LIN {X 0,Y 516.034,Z 964.883,A -85,B 0,C 180,E1 13801.811,E2 13801.811} C_VEL
LIN {X 0,Y 525.907,Z 921.872,A -85,B 0,C 180,E1 13804.841,E2 13804.841} C_VEL
LIN {X 0,Y 533.905,Z 879.595,A -85,B 0,C 180,E1 13807.015,E2 13807.015} C_VEL
LIN {X 0,Y 536.579,Z 858.24,A -85,B 0,C 180,E1 13807.941,E2 13807.941} C_VEL
LIN {X 0,Y 518.339,Z 819.478,A -85,B 0,C 180,E1 13812.064,E2 13812.064} C_VEL
LIN {X 0,Y 498.945,Z 786.831,A -85,B 0,C 180,E1 13816.041,E2 13816.041} C_VEL
LIN {X 0,Y 481.398,Z 761.941,A -85,B 0,C 180,E1 13819.773,E2 13819.773} C_VEL
LIN {X 0,Y 477.173,Z 755.892,A -85,B 0,C 180,E1 13820.762,E2 13820.762} C_VEL
LIN {X 0,Y 474.157,Z 751.123,A -85,B 0,C 180,E1 13821.51,E2 13821.51} C_VEL
LIN {X 0,Y 474.006,Z 749.56,A -85,B 0,C 180,E1 13821.607,E2 13821.607} C_VEL
LIN {X 0,Y 473.918,Z 749.56,A -85,B 0,C 180,E1 13827.169,E2 13827.169} C_VEL
LIN {X 0,Y 474.069,Z 749.56,A -85,B 0,C 180,E1 13833.49,E2 13833.49} C_VEL
LIN {X 0,Y 474.276,Z 749.56,A -85,B 0,C 180,E1 13839.477,E2 13839.477} C_VEL
LIN {X 0,Y 474.538,Z 749.56,A -85,B 0,C 180,E1 13845.235,E2 13845.235} C_VEL
LIN {X 0,Y 475.007,Z 749.56,A -85,B 0,C 180,E1 13850.842,E2 13850.842} C_VEL
LIN {X 0,Y 475.371,Z 749.56,A -85,B 0,C 180,E1 13856.35,E2 13856.35} C_VEL
LIN {X 0,Y 475.462,Z 749.56,A -85,B 0,C 180,E1 13861.816,E2 13861.816} C_VEL
LIN {X 0,Y 475.102,Z 749.56,A -85,B 0,C 180,E1 13867.304,E2 13867.304} C_VEL
LIN {X 0,Y 474.846,Z 749.56,A -85,B 0,C 180,E1 13872.867,E2 13872.867} C_VEL
LIN {X 0,Y 474.618,Z 749.56,A -85,B 0,C 180,E1 13878.561,E2 13878.561} C_VEL
LIN {X 0,Y 474.385,Z 750.237,A -85,B 0,C 180,E1 13884.27,E2 13884.27} C_VEL
LIN {X 0,Y 477.004,Z 755.483,A -85,B 0,C 180,E1 13884.954,E2 13884.954} C_VEL
LIN {X 0,Y 479.513,Z 758.583,A -85,B 0,C 180,E1 13885.535,E2 13885.535} C_VEL
LIN {X 0,Y 500.029,Z 787.996,A -85,B 0,C 180,E1 13889.906,E2 13889.906} C_VEL
LIN {X 0,Y 523.015,Z 825.421,A -85,B 0,C 180,E1 13894.162,E2 13894.162} C_VEL
LIN {X 0,Y 542.914,Z 863.835,A -85,B 0,C 180,E1 13897.881,E2 13897.881} C_VEL
LIN {X 0,Y 544.784,Z 869.388,A -85,B 0,C 180,E1 13898.295,E2 13898.295} C_VEL
LIN {X 0,Y 537.645,Z 917.442,A -85,B 0,C 180,E1 13899.901,E2 13899.901} C_VEL
LIN {X 0,Y 529.329,Z 963.938,A -85,B 0,C 180,E1 13902.158,E2 13902.158} C_VEL
LIN {X 0,Y 519.683,Z 1007.812,A -85,B 0,C 180,E1 13905.042,E2 13905.042} C_VEL
LIN {X 0,Y 509.605,Z 1048.714,A -85,B 0,C 180,E1 13908.52,E2 13908.52} C_VEL
LIN {X 0,Y 499.79,Z 1087.044,A -85,B 0,C 180,E1 13912.791,E2 13912.791} C_VEL
LIN {X 0,Y 491.205,Z 1120.824,A -85,B 0,C 180,E1 13917.595,E2 13917.595} C_VEL
LIN {X 0,Y 484.254,Z 1149.865,A -85,B 0,C 180,E1 13922.926,E2 13922.926} C_VEL
LIN {X 0,Y 479.949,Z 1171.932,A -85,B 0,C 180,E1 13928.124,E2 13928.124} C_VEL
LIN {X 0,Y 477.25,Z 1188.833,A -85,B 0,C 180,E1 13933.442,E2 13933.442} C_VEL
LIN {X 0,Y 475.934,Z 1200.642,A -85,B 0,C 180,E1 13939.017,E2 13939.017} C_VEL
LIN {X 0,Y 475.666,Z 1203.715,A -85,B 0,C 180,E1 13941.011,E2 13941.011} C_VEL
LIN {X 0,Y 473.053,Z 1205.774,A -85,B 0,C 180,E1 13942.541,E2 13942.541} C_VEL
LIN {X 0,Y 467.534,Z 1208.179,A -85,B 0,C 180,E1 13945.048,E2 13945.048} C_VEL
LIN {X 0,Y 467.525,Z 1208.086,A -85,B 0,C 180,E1 13945.115,E2 13945.115} C_VEL
LIN {X 0,Y 467.648,Z 1210,A -85,B 0,C 180,E1 13949.999,E2 13949.999} C_VEL
LIN {X 0,Y 467.584,Z 1207.633,A -85,B 0,C 180,E1 13955.563,E2 13955.563} C_VEL
LIN {X 0,Y 468.047,Z 1200.643,A -85,B 0,C 180,E1 13961.169,E2 13961.169} C_VEL
LIN {X 0,Y 469.297,Z 1189.506,A -85,B 0,C 180,E1 13966.364,E2 13966.364} C_VEL
LIN {X 0,Y 471.984,Z 1172.687,A -85,B 0,C 180,E1 13971.811,E2 13971.811} C_VEL
LIN {X 0,Y 476.377,Z 1150.561,A -85,B 0,C 180,E1 13977.183,E2 13977.183} C_VEL
LIN {X 0,Y 483.69,Z 1120.879,A -85,B 0,C 180,E1 13982.724,E2 13982.724} C_VEL
LIN {X 0,Y 492.65,Z 1086.82,A -85,B 0,C 180,E1 13987.664,E2 13987.664} C_VEL
LIN {X 0,Y 503.17,Z 1048.376,A -85,B 0,C 180,E1 13992.052,E2 13992.052} C_VEL
LIN {X 0,Y 514.127,Z 1007.233,A -85,B 0,C 180,E1 13995.657,E2 13995.657} C_VEL
LIN {X 0,Y 524.703,Z 963.33,A -85,B 0,C 180,E1 13998.628,E2 13998.628} C_VEL
LIN {X 0,Y 534.281,Z 915.858,A -85,B 0,C 180,E1 14000.977,E2 14000.977} C_VEL
LIN {X 0,Y 541.086,Z 870.88,A -85,B 0,C 180,E1 14002.601,E2 14002.601} C_VEL
LIN {X 0,Y 528.086,Z 840.131,A -85,B 0,C 180,E1 14005.85,E2 14005.85} C_VEL
LIN {X 0,Y 513.151,Z 814.352,A -85,B 0,C 180,E1 14009.429,E2 14009.429} C_VEL
LIN {X 0,Y 497.416,Z 791.232,A -85,B 0,C 180,E1 14013.626,E2 14013.626} C_VEL
LIN {X 0,Y 486.968,Z 777.414,A -85,B 0,C 180,E1 14016.94,E2 14016.94} C_VEL
LIN {X 0,Y 482.346,Z 771.07,A -85,B 0,C 180,E1 14018.647,E2 14018.647} C_VEL
LIN {X 0,Y 478.295,Z 764.996,A -85,B 0,C 180,E1 14020.33,E2 14020.33} C_VEL
LIN {X 0,Y 473.236,Z 759.393,A -85,B 0,C 180,E1 14022.628,E2 14022.628} C_VEL
LIN {X 0,Y 472.102,Z 757.06,A -85,B 0,C 180,E1 14023.262,E2 14023.262} C_VEL
LIN {X 0,Y 467.454,Z 752.711,A -85,B 0,C 180,E1 14025.88,E2 14025.88} C_VEL
LIN {X 0,Y 466.84,Z 749.56,A -85,B 0,C 180,E1 14026.622,E2 14026.622} C_VEL
LIN {X 0,Y 467.194,Z 749.56,A -85,B 0,C 180,E1 14032.571,E2 14032.571} C_VEL
LIN {X 0,Y 467.541,Z 749.56,A -85,B 0,C 180,E1 14038.153,E2 14038.153} C_VEL
LIN {X 0,Y 467.467,Z 749.56,A -85,B 0,C 180,E1 14043.712,E2 14043.712} C_VEL
LIN {X 0,Y 467.127,Z 750.157,A -85,B 0,C 180,E1 14049.255,E2 14049.255} C_VEL
LIN {X 0,Y 469.125,Z 754.964,A -85,B 0,C 180,E1 14050.679,E2 14050.679} C_VEL
LIN {X 0,Y 472.981,Z 758.131,A -85,B 0,C 180,E1 14052.694,E2 14052.694} C_VEL
LIN {X 0,Y 476.564,Z 763.704,A -85,B 0,C 180,E1 14054.466,E2 14054.466} C_VEL
LIN {X 0,Y 478.873,Z 766.162,A -85,B 0,C 180,E1 14055.447,E2 14055.447} C_VEL
LIN {X 0,Y 483.501,Z 771.831,A -85,B 0,C 180,E1 14057.278,E2 14057.278} C_VEL
LIN {X 0,Y 495.775,Z 789.143,A -85,B 0,C 180,E1 14061.46,E2 14061.46} C_VEL
LIN {X 0,Y 509.693,Z 809.728,A -85,B 0,C 180,E1 14065.505,E2 14065.505} C_VEL
LIN {X 0,Y 524.946,Z 837.122,A -85,B 0,C 180,E1 14069.707,E2 14069.707} C_VEL
LIN {X 0,Y 536.072,Z 863.906,A -85,B 0,C 180,E1 14073.041,E2 14073.041} C_VEL
LIN {X 0,Y 527.801,Z 907.851,A -85,B 0,C 180,E1 14075.105,E2 14075.105} C_VEL
LIN {X 0,Y 517.224,Z 951.582,A -85,B 0,C 180,E1 14077.925,E2 14077.925} C_VEL
LIN {X 0,Y 506.236,Z 989.958,A -85,B 0,C 180,E1 14081.275,E2 14081.275} C_VEL
LIN {X 0,Y 495.534,Z 1024.827,A -85,B 0,C 180,E1 14085.28,E2 14085.28} C_VEL
LIN {X 0,Y 485.435,Z 1057.02,A -85,B 0,C 180,E1 14090.171,E2 14090.171} C_VEL
LIN {X 0,Y 477.545,Z 1083.26,A -85,B 0,C 180,E1 14095.49,E2 14095.49} C_VEL
LIN {X 0,Y 472.449,Z 1103.182,A -85,B 0,C 180,E1 14100.863,E2 14100.863} C_VEL
LIN {X 0,Y 469.435,Z 1118.79,A -85,B 0,C 180,E1 14106.773,E2 14106.773} C_VEL
LIN {X 0,Y 468.084,Z 1127.979,A -85,B 0,C 180,E1 14112.018,E2 14112.018} C_VEL
LIN {X 0,Y 467.456,Z 1132.689,A -85,B 0,C 180,E1 14116.922,E2 14116.922} C_VEL
LIN {X 0,Y 467.499,Z 1133.645,A -85,B 0,C 180,E1 14122.572,E2 14122.572} C_VEL
LIN {X 0,Y 467.96,Z 1129.93,A -85,B 0,C 180,E1 14128.15,E2 14128.15} C_VEL
LIN {X 0,Y 468.682,Z 1123.231,A -85,B 0,C 180,E1 14132.773,E2 14132.773} C_VEL
LIN {X 0,Y 470.731,Z 1110.667,A -85,B 0,C 180,E1 14138.307,E2 14138.307} C_VEL
LIN {X 0,Y 474.702,Z 1092.283,A -85,B 0,C 180,E1 14143.95,E2 14143.95} C_VEL
LIN {X 0,Y 481.275,Z 1067.827,A -85,B 0,C 180,E1 14149.426,E2 14149.426} C_VEL
LIN {X 0,Y 489.77,Z 1038.333,A -85,B 0,C 180,E1 14154.336,E2 14154.336} C_VEL
LIN {X 0,Y 498.722,Z 1007.255,A -85,B 0,C 180,E1 14158.332,E2 14158.332} C_VEL
LIN {X 0,Y 509.579,Z 966.995,A -85,B 0,C 180,E1 14162.262,E2 14162.262} C_VEL
LIN {X 0,Y 519.366,Z 925.891,A -85,B 0,C 180,E1 14165.223,E2 14165.223} C_VEL
LIN {X 0,Y 527.743,Z 884.022,A -85,B 0,C 180,E1 14167.459,E2 14167.459} C_VEL
LIN {X 0,Y 530.718,Z 861.648,A -85,B 0,C 180,E1 14168.452,E2 14168.452} C_VEL
LIN {X 0,Y 512.892,Z 823.196,A -85,B 0,C 180,E1 14172.661,E2 14172.661} C_VEL
LIN {X 0,Y 494.247,Z 791.316,A -85,B 0,C 180,E1 14176.677,E2 14176.677} C_VEL
LIN {X 0,Y 474.619,Z 762.94,A -85,B 0,C 180,E1 14181.073,E2 14181.073} C_VEL
LIN {X 0,Y 469.179,Z 755.865,A -85,B 0,C 180,E1 14182.418,E2 14182.418} C_VEL
LIN {X 0,Y 466.211,Z 751.36,A -85,B 0,C 180,E1 14183.207,E2 14183.207} C_VEL
LIN {X 0,Y 465.989,Z 749.56,A -85,B 0,C 180,E1 14183.452,E2 14183.452} C_VEL
LIN {X 0,Y 466.023,Z 749.56,A -85,B 0,C 180,E1 14188.74,E2 14188.74} C_VEL
LIN {X 0,Y 466.202,Z 749.56,A -85,B 0,C 180,E1 14195.175,E2 14195.175} C_VEL
LIN {X 0,Y 466.369,Z 749.56,A -85,B 0,C 180,E1 14201.088,E2 14201.088} C_VEL
LIN {X 0,Y 466.749,Z 749.56,A -85,B 0,C 180,E1 14206.896,E2 14206.896} C_VEL
LIN {X 0,Y 467.16,Z 749.56,A -85,B 0,C 180,E1 14213.134,E2 14213.134} C_VEL
LIN {X 0,Y 467.5,Z 749.56,A -85,B 0,C 180,E1 14218.143,E2 14218.143} C_VEL
LIN {X 0,Y 467.378,Z 749.56,A -85,B 0,C 180,E1 14223.703,E2 14223.703} C_VEL
LIN {X 0,Y 467.105,Z 749.56,A -85,B 0,C 180,E1 14229.304,E2 14229.304} C_VEL
LIN {X 0,Y 466.815,Z 749.56,A -85,B 0,C 180,E1 14235.004,E2 14235.004} C_VEL
LIN {X 0,Y 466.573,Z 749.56,A -85,B 0,C 180,E1 14240.866,E2 14240.866} C_VEL
LIN {X 0,Y 466.512,Z 749.56,A -85,B 0,C 180,E1 14242.549,E2 14242.549} C_VEL
LIN {X 0,Y 468.426,Z 754.764,A -85,B 0,C 180,E1 14243.147,E2 14243.147} C_VEL
LIN {X 0,Y 471.571,Z 758.169,A -85,B 0,C 180,E1 14243.922,E2 14243.922} C_VEL
LIN {X 0,Y 490.297,Z 784.992,A -85,B 0,C 180,E1 14248.218,E2 14248.218} C_VEL
LIN {X 0,Y 513.116,Z 820.927,A -85,B 0,C 180,E1 14252.694,E2 14252.694} C_VEL
LIN {X 0,Y 535.57,Z 863.511,A -85,B 0,C 180,E1 14257.025,E2 14257.025} C_VEL
LIN {X 0,Y 539.079,Z 871.267,A -85,B 0,C 180,E1 14257.741,E2 14257.741} C_VEL
LIN {X 0,Y 531.631,Z 919.66,A -85,B 0,C 180,E1 14259.391,E2 14259.391} C_VEL
LIN {X 0,Y 523.197,Z 964.81,A -85,B 0,C 180,E1 14261.624,E2 14261.624} C_VEL
LIN {X 0,Y 513.294,Z 1008.41,A -85,B 0,C 180,E1 14264.526,E2 14264.526} C_VEL
LIN {X 0,Y 503.16,Z 1048.159,A -85,B 0,C 180,E1 14267.939,E2 14267.939} C_VEL
LIN {X 0,Y 492.821,Z 1087.152,A -85,B 0,C 180,E1 14272.33,E2 14272.33} C_VEL
LIN {X 0,Y 484.096,Z 1119.989,A -85,B 0,C 180,E1 14277.054,E2 14277.054} C_VEL
LIN {X 0,Y 476.795,Z 1149.453,A -85,B 0,C 180,E1 14282.542,E2 14282.542} C_VEL
LIN {X 0,Y 472.213,Z 1171.658,A -85,B 0,C 180,E1 14287.866,E2 14287.866} C_VEL
LIN {X 0,Y 469.29,Z 1189.515,A -85,B 0,C 180,E1 14293.634,E2 14293.634} C_VEL
LIN {X 0,Y 468.056,Z 1200.64,A -85,B 0,C 180,E1 14298.83,E2 14298.83} C_VEL
LIN {X 0,Y 467.59,Z 1207.63,A -85,B 0,C 180,E1 14304.435,E2 14304.435} C_VEL
LIN {X 0,Y 467.525,Z 1208.086,A -85,B 0,C 180,E1 14305.115,E2 14305.115} C_VEL
LIN {X 0,Y 466.231,Z 1208.813,A -85,B 0,C 180,E1 14306.171,E2 14306.171} C_VEL
LIN {X 0,Y 459.71,Z 1209.836,A -85,B 0,C 180,E1 14309.058,E2 14309.058} C_VEL
LIN {X 0,Y 459.645,Z 1209.881,A -85,B 0,C 180,E1 14309.332,E2 14309.332} C_VEL
LIN {X 0,Y 459.669,Z 1208.874,A -85,B 0,C 180,E1 14313.769,E2 14313.769} C_VEL
LIN {X 0,Y 459.894,Z 1204.643,A -85,B 0,C 180,E1 14318.502,E2 14318.502} C_VEL
LIN {X 0,Y 460.731,Z 1194.895,A -85,B 0,C 180,E1 14324.087,E2 14324.087} C_VEL
LIN {X 0,Y 463.058,Z 1179.167,A -85,B 0,C 180,E1 14330.038,E2 14330.038} C_VEL
LIN {X 0,Y 467.242,Z 1157.503,A -85,B 0,C 180,E1 14335.886,E2 14335.886} C_VEL
LIN {X 0,Y 473.839,Z 1130.433,A -85,B 0,C 180,E1 14341.48,E2 14341.48} C_VEL
LIN {X 0,Y 483.134,Z 1096.017,A -85,B 0,C 180,E1 14346.934,E2 14346.934} C_VEL
LIN {X 0,Y 493.624,Z 1059.485,A -85,B 0,C 180,E1 14351.454,E2 14351.454} C_VEL
LIN {X 0,Y 505.554,Z 1017.069,A -85,B 0,C 180,E1 14355.501,E2 14355.501} C_VEL
LIN {X 0,Y 516.733,Z 973.238,A -85,B 0,C 180,E1 14358.679,E2 14358.679} C_VEL
LIN {X 0,Y 527.419,Z 925.022,A -85,B 0,C 180,E1 14361.262,E2 14361.262} C_VEL
LIN {X 0,Y 535.794,Z 874.352,A -85,B 0,C 180,E1 14363.158,E2 14363.158} C_VEL
LIN {X 0,Y 523.909,Z 845.325,A -85,B 0,C 180,E1 14366.338,E2 14366.338} C_VEL
LIN {X 0,Y 509.157,Z 819.264,A -85,B 0,C 180,E1 14370.06,E2 14370.06} C_VEL
LIN {X 0,Y 494.374,Z 797.334,A -85,B 0,C 180,E1 14374.176,E2 14374.176} C_VEL
LIN {X 0,Y 484.785,Z 784.4,A -85,B 0,C 180,E1 14377.315,E2 14377.315} C_VEL
LIN {X 0,Y 480.104,Z 778.097,A -85,B 0,C 180,E1 14379.086,E2 14379.086} C_VEL
LIN {X 0,Y 475.37,Z 771.607,A -85,B 0,C 180,E1 14381.109,E2 14381.109} C_VEL
LIN {X 0,Y 471.196,Z 765.717,A -85,B 0,C 180,E1 14383.169,E2 14383.169} C_VEL
LIN {X 0,Y 465.66,Z 759.194,A -85,B 0,C 180,E1 14386.444,E2 14386.444} C_VEL
LIN {X 0,Y 465.212,Z 757.285,A -85,B 0,C 180,E1 14386.862,E2 14386.862} C_VEL
LIN {X 0,Y 459.754,Z 752.456,A -85,B 0,C 180,E1 14391.753,E2 14391.753} C_VEL
LIN {X 0,Y 459.295,Z 749.56,A -85,B 0,C 180,E1 14392.918,E2 14392.918} C_VEL
LIN {X 0,Y 459.632,Z 749.56,A -85,B 0,C 180,E1 14398.121,E2 14398.121} C_VEL
LIN {X 0,Y 459.572,Z 750.284,A -85,B 0,C 180,E1 14403.186,E2 14403.186} C_VEL
LIN {X 0,Y 462.259,Z 755.712,A -85,B 0,C 180,E1 14406.457,E2 14406.457} C_VEL
LIN {X 0,Y 465.72,Z 758.308,A -85,B 0,C 180,E1 14409.027,E2 14409.027} C_VEL
LIN {X 0,Y 468.761,Z 763.51,A -85,B 0,C 180,E1 14411.04,E2 14411.04} C_VEL
LIN {X 0,Y 471.522,Z 766.138,A -85,B 0,C 180,E1 14412.499,E2 14412.499} C_VEL
LIN {X 0,Y 475.727,Z 771.71,A -85,B 0,C 180,E1 14414.54,E2 14414.54} C_VEL
LIN {X 0,Y 483.141,Z 781.942,A -85,B 0,C 180,E1 14417.585,E2 14417.585} C_VEL
LIN {X 0,Y 492.503,Z 794.697,A -85,B 0,C 180,E1 14420.843,E2 14420.843} C_VEL
LIN {X 0,Y 507.227,Z 817.31,A -85,B 0,C 180,E1 14425.337,E2 14425.337} C_VEL
LIN {X 0,Y 521.417,Z 844.31,A -85,B 0,C 180,E1 14429.523,E2 14429.523} C_VEL
LIN {X 0,Y 530.931,Z 868.507,A -85,B 0,C 180,E1 14432.561,E2 14432.561} C_VEL
LIN {X 0,Y 522.001,Z 911.598,A -85,B 0,C 180,E1 14434.611,E2 14434.611} C_VEL
LIN {X 0,Y 511.337,Z 953.906,A -85,B 0,C 180,E1 14437.4,E2 14437.4} C_VEL
LIN {X 0,Y 499.675,Z 993.02,A -85,B 0,C 180,E1 14440.884,E2 14440.884} C_VEL
LIN {X 0,Y 489.157,Z 1025.801,A -85,B 0,C 180,E1 14444.723,E2 14444.723} C_VEL
LIN {X 0,Y 478.492,Z 1058.247,A -85,B 0,C 180,E1 14449.721,E2 14449.721} C_VEL
LIN {X 0,Y 470.071,Z 1084.955,A -85,B 0,C 180,E1 14455.262,E2 14455.262} C_VEL
LIN {X 0,Y 464.702,Z 1104.813,A -85,B 0,C 180,E1 14460.807,E2 14460.807} C_VEL
LIN {X 0,Y 461.574,Z 1120.275,A -85,B 0,C 180,E1 14466.868,E2 14466.868} C_VEL
LIN {X 0,Y 460.107,Z 1129.764,A -85,B 0,C 180,E1 14472.808,E2 14472.808} C_VEL
LIN {X 0,Y 459.545,Z 1134.222,A -85,B 0,C 180,E1 14478.622,E2 14478.622} C_VEL
LIN {X 0,Y 459.74,Z 1133.619,A -85,B 0,C 180,E1 14484.342,E2 14484.342} C_VEL
LIN {X 0,Y 460.402,Z 1128.5,A -85,B 0,C 180,E1 14490.001,E2 14490.001} C_VEL
LIN {X 0,Y 461.723,Z 1118.545,A -85,B 0,C 180,E1 14495.636,E2 14495.636} C_VEL
LIN {X 0,Y 464.674,Z 1103.6,A -85,B 0,C 180,E1 14501.253,E2 14501.253} C_VEL
LIN {X 0,Y 469.925,Z 1082.798,A -85,B 0,C 180,E1 14506.824,E2 14506.824} C_VEL
LIN {X 0,Y 477.715,Z 1056.501,A -85,B 0,C 180,E1 14512.065,E2 14512.065} C_VEL
LIN {X 0,Y 487.558,Z 1023.793,A -85,B 0,C 180,E1 14516.956,E2 14516.956} C_VEL
LIN {X 0,Y 497.86,Z 988.391,A -85,B 0,C 180,E1 14520.938,E2 14520.938} C_VEL
LIN {X 0,Y 507.844,Z 950.913,A -85,B 0,C 180,E1 14524.17,E2 14524.17} C_VEL
LIN {X 0,Y 517.899,Z 906.495,A -85,B 0,C 180,E1 14527,E2 14527} C_VEL
LIN {X 0,Y 525.227,Z 866.927,A -85,B 0,C 180,E1 14528.829,E2 14528.829} C_VEL
LIN {X 0,Y 510.404,Z 832.701,A -85,B 0,C 180,E1 14532.602,E2 14532.602} C_VEL
LIN {X 0,Y 492.456,Z 800.032,A -85,B 0,C 180,E1 14536.707,E2 14536.707} C_VEL
LIN {X 0,Y 471.991,Z 769.876,A -85,B 0,C 180,E1 14541.408,E2 14541.408} C_VEL
LIN {X 0,Y 463.065,Z 757.342,A -85,B 0,C 180,E1 14543.731,E2 14543.731} C_VEL
LIN {X 0,Y 458.341,Z 751.881,A -85,B 0,C 180,E1 14545.03,E2 14545.03} C_VEL
LIN {X 0,Y 458.001,Z 749.56,A -85,B 0,C 180,E1 14545.26,E2 14545.26} C_VEL
LIN {X 0,Y 458.11,Z 749.56,A -85,B 0,C 180,E1 14550.337,E2 14550.337} C_VEL
LIN {X 0,Y 458.29,Z 749.56,A -85,B 0,C 180,E1 14556.685,E2 14556.685} C_VEL
LIN {X 0,Y 458.563,Z 749.56,A -85,B 0,C 180,E1 14562.876,E2 14562.876} C_VEL
LIN {X 0,Y 459.016,Z 749.56,A -85,B 0,C 180,E1 14568.602,E2 14568.602} C_VEL
LIN {X 0,Y 459.376,Z 749.56,A -85,B 0,C 180,E1 14574.331,E2 14574.331} C_VEL
LIN {X 0,Y 459.778,Z 749.56,A -85,B 0,C 180,E1 14579.995,E2 14579.995} C_VEL
LIN {X 0,Y 459.434,Z 749.56,A -85,B 0,C 180,E1 14585.658,E2 14585.658} C_VEL
LIN {X 0,Y 459.063,Z 749.56,A -85,B 0,C 180,E1 14591.386,E2 14591.386} C_VEL
LIN {X 0,Y 458.841,Z 749.56,A -85,B 0,C 180,E1 14597.237,E2 14597.237} C_VEL
LIN {X 0,Y 458.695,Z 749.792,A -85,B 0,C 180,E1 14600.743,E2 14600.743} C_VEL
LIN {X 0,Y 460.705,Z 754.891,A -85,B 0,C 180,E1 14601.398,E2 14601.398} C_VEL
LIN {X 0,Y 463.893,Z 758.355,A -85,B 0,C 180,E1 14602.252,E2 14602.252} C_VEL
LIN {X 0,Y 482.485,Z 784.523,A -85,B 0,C 180,E1 14606.816,E2 14606.816} C_VEL
LIN {X 0,Y 503.927,Z 817.831,A -85,B 0,C 180,E1 14611.271,E2 14611.271} C_VEL
LIN {X 0,Y 526.471,Z 859.855,A -85,B 0,C 180,E1 14615.791,E2 14615.791} C_VEL
LIN {X 0,Y 533.205,Z 874.662,A -85,B 0,C 180,E1 14617.22,E2 14617.22} C_VEL
LIN {X 0,Y 525.724,Z 921.347,A -85,B 0,C 180,E1 14618.849,E2 14618.849} C_VEL
LIN {X 0,Y 517.009,Z 966.045,A -85,B 0,C 180,E1 14621.101,E2 14621.101} C_VEL
LIN {X 0,Y 506.432,Z 1011.027,A -85,B 0,C 180,E1 14624.151,E2 14624.151} C_VEL
LIN {X 0,Y 495.77,Z 1051.039,A -85,B 0,C 180,E1 14627.697,E2 14627.697} C_VEL
LIN {X 0,Y 484.932,Z 1090.594,A -85,B 0,C 180,E1 14632.285,E2 14632.285} C_VEL
LIN {X 0,Y 476.14,Z 1122.387,A -85,B 0,C 180,E1 14637.055,E2 14637.055} C_VEL
LIN {X 0,Y 468.748,Z 1151.201,A -85,B 0,C 180,E1 14642.602,E2 14642.602} C_VEL
LIN {X 0,Y 464.329,Z 1172.068,A -85,B 0,C 180,E1 14647.81,E2 14647.81} C_VEL
LIN {X 0,Y 461.506,Z 1188.835,A -85,B 0,C 180,E1 14653.35,E2 14653.35} C_VEL
LIN {X 0,Y 460.184,Z 1200.257,A -85,B 0,C 180,E1 14658.636,E2 14658.636} C_VEL
LIN {X 0,Y 459.825,Z 1205.885,A -85,B 0,C 180,E1 14662.446,E2 14662.446} C_VEL
LIN {X 0,Y 459.621,Z 1209.665,A -85,B 0,C 180,E1 14668.115,E2 14668.115} C_VEL
LIN {X 0,Y 459.645,Z 1209.881,A -85,B 0,C 180,E1 14669.332,E2 14669.332} C_VEL
LIN {X 0,Y 457.208,Z 1209.872,A -85,B 0,C 180,E1 14670.944,E2 14670.944} C_VEL
LIN {X 0,Y 451.866,Z 1208.739,A -85,B 0,C 180,E1 14673.363,E2 14673.363} C_VEL
LIN {X 0,Y 451.776,Z 1208.547,A -85,B 0,C 180,E1 14673.643,E2 14673.643} C_VEL
LIN {X 0,Y 452.009,Z 1203.973,A -85,B 0,C 180,E1 14678.652,E2 14678.652} C_VEL
LIN {X 0,Y 453.001,Z 1193.447,A -85,B 0,C 180,E1 14684.689,E2 14684.689} C_VEL
LIN {X 0,Y 455.344,Z 1178.421,A -85,B 0,C 180,E1 14690.392,E2 14690.392} C_VEL
LIN {X 0,Y 459.757,Z 1156.693,A -85,B 0,C 180,E1 14696.34,E2 14696.34} C_VEL
LIN {X 0,Y 466.853,Z 1129.074,A -85,B 0,C 180,E1 14702.117,E2 14702.117} C_VEL
LIN {X 0,Y 476.541,Z 1095.135,A -85,B 0,C 180,E1 14707.562,E2 14707.562} C_VEL
LIN {X 0,Y 487.373,Z 1058.993,A -85,B 0,C 180,E1 14712.088,E2 14712.088} C_VEL
LIN {X 0,Y 499.595,Z 1017.17,A -85,B 0,C 180,E1 14716.125,E2 14716.125} C_VEL
LIN {X 0,Y 510.729,Z 975.412,A -85,B 0,C 180,E1 14719.206,E2 14719.206} C_VEL
LIN {X 0,Y 521.995,Z 926.551,A -85,B 0,C 180,E1 14721.866,E2 14721.866} C_VEL
LIN {X 0,Y 530.615,Z 877.923,A -85,B 0,C 180,E1 14723.714,E2 14723.714} C_VEL
LIN {X 0,Y 519.298,Z 849.736,A -85,B 0,C 180,E1 14726.909,E2 14726.909} C_VEL
LIN {X 0,Y 504.536,Z 823.025,A -85,B 0,C 180,E1 14730.886,E2 14730.886} C_VEL
LIN {X 0,Y 488.77,Z 799.383,A -85,B 0,C 180,E1 14735.582,E2 14735.582} C_VEL
LIN {X 0,Y 478.312,Z 785.472,A -85,B 0,C 180,E1 14739.367,E2 14739.367} C_VEL
LIN {X 0,Y 473.411,Z 778.834,A -85,B 0,C 180,E1 14741.511,E2 14741.511} C_VEL
LIN {X 0,Y 468.417,Z 772.017,A -85,B 0,C 180,E1 14744.09,E2 14744.09} C_VEL
LIN {X 0,Y 464.127,Z 766.28,A -85,B 0,C 180,E1 14746.831,E2 14746.831} C_VEL
LIN {X 0,Y 462.589,Z 764.591,A -85,B 0,C 180,E1 14747.974,E2 14747.974} C_VEL
LIN {X 0,Y 458.345,Z 758.989,A -85,B 0,C 180,E1 14752.487,E2 14752.487} C_VEL
LIN {X 0,Y 457.931,Z 757.318,A -85,B 0,C 180,E1 14753.373,E2 14753.373} C_VEL
LIN {X 0,Y 458.42,Z 757.813,A -85,B 0,C 180,E1 14762.899,E2 14762.899} C_VEL
LIN {X 0,Y 460.897,Z 763.289,A -85,B 0,C 180,E1 14766.122,E2 14766.122} C_VEL
LIN {X 0,Y 464.341,Z 766.044,A -85,B 0,C 180,E1 14768.779,E2 14768.779} C_VEL
LIN {X 0,Y 468.01,Z 771.628,A -85,B 0,C 180,E1 14771.176,E2 14771.176} C_VEL
LIN {X 0,Y 470.042,Z 773.858,A -85,B 0,C 180,E1 14772.273,E2 14772.273} C_VEL
LIN {X 0,Y 475.956,Z 782.104,A -85,B 0,C 180,E1 14775.131,E2 14775.131} C_VEL
LIN {X 0,Y 481.613,Z 789.905,A -85,B 0,C 180,E1 14777.465,E2 14777.465} C_VEL
LIN {X 0,Y 490.45,Z 802.199,A -85,B 0,C 180,E1 14780.616,E2 14780.616} C_VEL
LIN {X 0,Y 504.273,Z 824.481,A -85,B 0,C 180,E1 14785.104,E2 14785.104} C_VEL
LIN {X 0,Y 517.567,Z 850.783,A -85,B 0,C 180,E1 14789.236,E2 14789.236} C_VEL
LIN {X 0,Y 525.638,Z 871.611,A -85,B 0,C 180,E1 14791.958,E2 14791.958} C_VEL
LIN {X 0,Y 515.666,Z 917.965,A -85,B 0,C 180,E1 14794.261,E2 14794.261} C_VEL
LIN {X 0,Y 504.82,Z 958.246,A -85,B 0,C 180,E1 14797.021,E2 14797.021} C_VEL
LIN {X 0,Y 492.782,Z 997.164,A -85,B 0,C 180,E1 14800.588,E2 14800.588} C_VEL
LIN {X 0,Y 480.701,Z 1032.84,A -85,B 0,C 180,E1 14804.992,E2 14804.992} C_VEL
LIN {X 0,Y 470.847,Z 1061.599,A -85,B 0,C 180,E1 14809.665,E2 14809.665} C_VEL
LIN {X 0,Y 462.171,Z 1088.305,A -85,B 0,C 180,E1 14815.429,E2 14815.429} C_VEL
LIN {X 0,Y 456.37,Z 1109.145,A -85,B 0,C 180,E1 14821.679,E2 14821.679} C_VEL
LIN {X 0,Y 453.505,Z 1122.596,A -85,B 0,C 180,E1 14827.469,E2 14827.469} C_VEL
LIN {X 0,Y 452.135,Z 1131.412,A -85,B 0,C 180,E1 14833.497,E2 14833.497} C_VEL
LIN {X 0,Y 451.683,Z 1134.809,A -85,B 0,C 180,E1 14838.421,E2 14838.421} C_VEL
LIN {X 0,Y 451.847,Z 1134.343,A -85,B 0,C 180,E1 14844.243,E2 14844.243} C_VEL
LIN {X 0,Y 452.565,Z 1129.316,A -85,B 0,C 180,E1 14850.001,E2 14850.001} C_VEL
LIN {X 0,Y 453.943,Z 1119.519,A -85,B 0,C 180,E1 14855.732,E2 14855.732} C_VEL
LIN {X 0,Y 456.98,Z 1104.679,A -85,B 0,C 180,E1 14861.445,E2 14861.445} C_VEL
LIN {X 0,Y 462.469,Z 1084.05,A -85,B 0,C 180,E1 14867.103,E2 14867.103} C_VEL
LIN {X 0,Y 470.524,Z 1057.949,A -85,B 0,C 180,E1 14872.42,E2 14872.42} C_VEL
LIN {X 0,Y 480.683,Z 1025.376,A -85,B 0,C 180,E1 14877.373,E2 14877.373} C_VEL
LIN {X 0,Y 491.003,Z 991.324,A -85,B 0,C 180,E1 14881.29,E2 14881.29} C_VEL
LIN {X 0,Y 501.55,Z 953.09,A -85,B 0,C 180,E1 14884.66,E2 14884.66} C_VEL
LIN {X 0,Y 511.48,Z 910.966,A -85,B 0,C 180,E1 14887.409,E2 14887.409} C_VEL
LIN {X 0,Y 519.229,Z 868.82,A -85,B 0,C 180,E1 14889.47,E2 14889.47} C_VEL
LIN {X 0,Y 502.783,Z 831.758,A -85,B 0,C 180,E1 14893.749,E2 14893.749} C_VEL
LIN {X 0,Y 485.076,Z 800.289,A -85,B 0,C 180,E1 14897.97,E2 14897.97} C_VEL
LIN {X 0,Y 467.804,Z 775.095,A -85,B 0,C 180,E1 14902.131,E2 14902.131} C_VEL
LIN {X 0,Y 458.718,Z 762.888,A -85,B 0,C 180,E1 14904.572,E2 14904.572} C_VEL
LIN {X 0,Y 454.18,Z 756.476,A -85,B 0,C 180,E1 14905.914,E2 14905.914} C_VEL
LIN {X 0,Y 450.488,Z 752.05,A -85,B 0,C 180,E1 14907.047,E2 14907.047} C_VEL
LIN {X 0,Y 450.086,Z 749.56,A -85,B 0,C 180,E1 14907.325,E2 14907.325} C_VEL
LIN {X 0,Y 450.31,Z 749.56,A -85,B 0,C 180,E1 14914.129,E2 14914.129} C_VEL
LIN {X 0,Y 450.499,Z 749.56,A -85,B 0,C 180,E1 14920.395,E2 14920.395} C_VEL
LIN {X 0,Y 450.904,Z 749.56,A -85,B 0,C 180,E1 14926.427,E2 14926.427} C_VEL
LIN {X 0,Y 451.343,Z 749.56,A -85,B 0,C 180,E1 14932.298,E2 14932.298} C_VEL
LIN {X 0,Y 451.709,Z 749.56,A -85,B 0,C 180,E1 14938.078,E2 14938.078} C_VEL
LIN {X 0,Y 451.559,Z 749.56,A -85,B 0,C 180,E1 14943.832,E2 14943.832} C_VEL
LIN {X 0,Y 451.242,Z 749.56,A -85,B 0,C 180,E1 14949.634,E2 14949.634} C_VEL
LIN {X 0,Y 450.942,Z 749.56,A -85,B 0,C 180,E1 14955.545,E2 14955.545} C_VEL
LIN {X 0,Y 450.825,Z 749.56,A -85,B 0,C 180,E1 14958.69,E2 14958.69} C_VEL
LIN {X 0,Y 452.798,Z 754.804,A -85,B 0,C 180,E1 14959.427,E2 14959.427} C_VEL
LIN {X 0,Y 456.148,Z 758.189,A -85,B 0,C 180,E1 14960.403,E2 14960.403} C_VEL
LIN {X 0,Y 474.768,Z 784.117,A -85,B 0,C 180,E1 14965.334,E2 14965.334} C_VEL
LIN {X 0,Y 495.891,Z 816.716,A -85,B 0,C 180,E1 14969.992,E2 14969.992} C_VEL
LIN {X 0,Y 515.98,Z 853.479,A -85,B 0,C 180,E1 14974.192,E2 14974.192} C_VEL
LIN {X 0,Y 527.372,Z 877.766,A -85,B 0,C 180,E1 14976.677,E2 14976.677} C_VEL
LIN {X 0,Y 519.657,Z 924.347,A -85,B 0,C 180,E1 14978.352,E2 14978.352} C_VEL
LIN {X 0,Y 510.428,Z 969.068,A -85,B 0,C 180,E1 14980.674,E2 14980.674} C_VEL
LIN {X 0,Y 499.973,Z 1012.104,A -85,B 0,C 180,E1 14983.651,E2 14983.651} C_VEL
LIN {X 0,Y 488.758,Z 1052.658,A -85,B 0,C 180,E1 14987.324,E2 14987.324} C_VEL
LIN {X 0,Y 478.095,Z 1090.271,A -85,B 0,C 180,E1 14991.755,E2 14991.755} C_VEL
LIN {X 0,Y 468.677,Z 1123.064,A -85,B 0,C 180,E1 14996.761,E2 14996.761} C_VEL
LIN {X 0,Y 461.043,Z 1151.74,A -85,B 0,C 180,E1 15002.405,E2 15002.405} C_VEL
LIN {X 0,Y 456.299,Z 1173.285,A -85,B 0,C 180,E1 15008.004,E2 15008.004} C_VEL
LIN {X 0,Y 453.375,Z 1190.6,A -85,B 0,C 180,E1 15014.038,E2 15014.038} C_VEL
LIN {X 0,Y 452.212,Z 1201.267,A -85,B 0,C 180,E1 15019.408,E2 15019.408} C_VEL
LIN {X 0,Y 451.793,Z 1207.113,A -85,B 0,C 180,E1 15024.24,E2 15024.24} C_VEL
LIN {X 0,Y 451.857,Z 1209.678,A -85,B 0,C 180,E1 15029.999,E2 15029.999} C_VEL
LIN {X 0,Y 451.776,Z 1208.547,A -85,B 0,C 180,E1 15033.643,E2 15033.643} C_VEL
LIN {X 0,Y 449.311,Z 1207.433,A -85,B 0,C 180,E1 15035.273,E2 15035.273} C_VEL
LIN {X 0,Y 444.147,Z 1204.728,A -85,B 0,C 180,E1 15037.707,E2 15037.707} C_VEL
LIN {X 0,Y 444.075,Z 1204.368,A -85,B 0,C 180,E1 15037.987,E2 15037.987} C_VEL
LIN {X 0,Y 444.83,Z 1195.234,A -85,B 0,C 180,E1 15043.756,E2 15043.756} C_VEL
LIN {X 0,Y 447.11,Z 1180.567,A -85,B 0,C 180,E1 15049.753,E2 15049.753} C_VEL
LIN {X 0,Y 451.385,Z 1160.056,A -85,B 0,C 180,E1 15055.797,E2 15055.797} C_VEL
LIN {X 0,Y 458.438,Z 1132.693,A -85,B 0,C 180,E1 15061.829,E2 15061.829} C_VEL
LIN {X 0,Y 467.415,Z 1102.471,A -85,B 0,C 180,E1 15067.022,E2 15067.022} C_VEL
LIN {X 0,Y 479.508,Z 1063.812,A -85,B 0,C 180,E1 15072.143,E2 15072.143} C_VEL
LIN {X 0,Y 491.34,Z 1025.273,A -85,B 0,C 180,E1 15076.067,E2 15076.067} C_VEL
LIN {X 0,Y 504.174,Z 979.81,A -85,B 0,C 180,E1 15079.602,E2 15079.602} C_VEL
LIN {X 0,Y 515.768,Z 932.163,A -85,B 0,C 180,E1 15082.283,E2 15082.283} C_VEL
LIN {X 0,Y 525.153,Z 884.394,A -85,B 0,C 180,E1 15084.179,E2 15084.179} C_VEL
LIN {X 0,Y 524.978,Z 880.155,A -85,B 0,C 180,E1 15084.433,E2 15084.433} C_VEL
LIN {X 0,Y 514.725,Z 854.195,A -85,B 0,C 180,E1 15087.483,E2 15087.483} C_VEL
LIN {X 0,Y 500.922,Z 828.77,A -85,B 0,C 180,E1 15091.404,E2 15091.404} C_VEL
LIN {X 0,Y 486.452,Z 806.367,A -85,B 0,C 180,E1 15095.939,E2 15095.939} C_VEL
LIN {X 0,Y 476.271,Z 792.533,A -85,B 0,C 180,E1 15099.76,E2 15099.76} C_VEL
LIN {X 0,Y 471.605,Z 786.123,A -85,B 0,C 180,E1 15101.861,E2 15101.861} C_VEL
LIN {X 0,Y 466.835,Z 779.546,A -85,B 0,C 180,E1 15104.396,E2 15104.396} C_VEL
LIN {X 0,Y 462.629,Z 773.412,A -85,B 0,C 180,E1 15107.208,E2 15107.208} C_VEL
LIN {X 0,Y 457.229,Z 766.652,A -85,B 0,C 180,E1 15112.707,E2 15112.707} C_VEL
LIN {X 0,Y 456.97,Z 765.141,A -85,B 0,C 180,E1 15113.359,E2 15113.359} C_VEL
LIN {X 0,Y 457.357,Z 765.738,A -85,B 0,C 180,E1 15122.787,E2 15122.787} C_VEL
LIN {X 0,Y 460.328,Z 771.517,A -85,B 0,C 180,E1 15126.485,E2 15126.485} C_VEL
LIN {X 0,Y 462.999,Z 773.758,A -85,B 0,C 180,E1 15128.545,E2 15128.545} C_VEL
LIN {X 0,Y 467.267,Z 779.69,A -85,B 0,C 180,E1 15131.312,E2 15131.312} C_VEL
LIN {X 0,Y 474.153,Z 789.436,A -85,B 0,C 180,E1 15134.836,E2 15134.836} C_VEL
LIN {X 0,Y 483.438,Z 802.295,A -85,B 0,C 180,E1 15138.633,E2 15138.633} C_VEL
LIN {X 0,Y 496.407,Z 823.031,A -85,B 0,C 180,E1 15143.251,E2 15143.251} C_VEL
LIN {X 0,Y 510.008,Z 848.935,A -85,B 0,C 180,E1 15147.742,E2 15147.742} C_VEL
LIN {X 0,Y 520.376,Z 875.341,A -85,B 0,C 180,E1 15151.398,E2 15151.398} C_VEL
LIN {X 0,Y 510.657,Z 918.774,A -85,B 0,C 180,E1 15153.576,E2 15153.576} C_VEL
LIN {X 0,Y 499.395,Z 959.254,A -85,B 0,C 180,E1 15156.369,E2 15156.369} C_VEL
LIN {X 0,Y 486.956,Z 998.06,A -85,B 0,C 180,E1 15159.953,E2 15159.953} C_VEL
LIN {X 0,Y 474.377,Z 1033.736,A -85,B 0,C 180,E1 15164.4,E2 15164.4} C_VEL
LIN {X 0,Y 464.186,Z 1062.113,A -85,B 0,C 180,E1 15169.062,E2 15169.062} C_VEL
LIN {X 0,Y 455.032,Z 1088.801,A -85,B 0,C 180,E1 15174.892,E2 15174.892} C_VEL
LIN {X 0,Y 448.989,Z 1109.161,A -85,B 0,C 180,E1 15181.066,E2 15181.066} C_VEL
LIN {X 0,Y 445.805,Z 1123.12,A -85,B 0,C 180,E1 15187.115,E2 15187.115} C_VEL
LIN {X 0,Y 444.334,Z 1131.911,A -85,B 0,C 180,E1 15193.198,E2 15193.198} C_VEL
LIN {X 0,Y 443.819,Z 1135.392,A -85,B 0,C 180,E1 15198.213,E2 15198.213} C_VEL
LIN {X 0,Y 443.836,Z 1135.669,A -85,B 0,C 180,E1 15202.174,E2 15202.174} C_VEL
LIN {X 0,Y 444.401,Z 1132.351,A -85,B 0,C 180,E1 15208.052,E2 15208.052} C_VEL
LIN {X 0,Y 445.184,Z 1125.987,A -85,B 0,C 180,E1 15212.919,E2 15212.919} C_VEL
LIN {X 0,Y 447.486,Z 1113.747,A -85,B 0,C 180,E1 15218.742,E2 15218.742} C_VEL
LIN {X 0,Y 451.762,Z 1096.699,A -85,B 0,C 180,E1 15224.431,E2 15224.431} C_VEL
LIN {X 0,Y 458.744,Z 1073.403,A -85,B 0,C 180,E1 15230.048,E2 15230.048} C_VEL
LIN {X 0,Y 467.803,Z 1045.706,A -85,B 0,C 180,E1 15235.07,E2 15235.07} C_VEL
LIN {X 0,Y 478.728,Z 1011.783,A -85,B 0,C 180,E1 15239.719,E2 15239.719} C_VEL
LIN {X 0,Y 489.744,Z 975.046,A -85,B 0,C 180,E1 15243.502,E2 15243.502} C_VEL
LIN {X 0,Y 500.437,Z 935.705,A -85,B 0,C 180,E1 15246.56,E2 15246.56} C_VEL
LIN {X 0,Y 509.814,Z 893.554,A -85,B 0,C 180,E1 15248.98,E2 15248.98} C_VEL
LIN {X 0,Y 513.561,Z 872.678,A -85,B 0,C 180,E1 15249.946,E2 15249.946} C_VEL
LIN {X 0,Y 497.821,Z 836.292,A -85,B 0,C 180,E1 15254.281,E2 15254.281} C_VEL
LIN {X 0,Y 481.61,Z 806.721,A -85,B 0,C 180,E1 15258.326,E2 15258.326} C_VEL
LIN {X 0,Y 464.803,Z 781.468,A -85,B 0,C 180,E1 15262.585,E2 15262.585} C_VEL
LIN {X 0,Y 455.668,Z 769.282,A -85,B 0,C 180,E1 15265.099,E2 15265.099} C_VEL
LIN {X 0,Y 451.065,Z 763.113,A -85,B 0,C 180,E1 15266.49,E2 15266.49} C_VEL
LIN {X 0,Y 446.352,Z 756.535,A -85,B 0,C 180,E1 15268.029,E2 15268.029} C_VEL
LIN {X 0,Y 442.603,Z 752.003,A -85,B 0,C 180,E1 15269.318,E2 15269.318} C_VEL
LIN {X 0,Y 442.293,Z 749.56,A -85,B 0,C 180,E1 15269.685,E2 15269.685} C_VEL
LIN {X 0,Y 442.396,Z 749.56,A -85,B 0,C 180,E1 15275.795,E2 15275.795} C_VEL
LIN {X 0,Y 442.642,Z 749.56,A -85,B 0,C 180,E1 15282.1,E2 15282.1} C_VEL
LIN {X 0,Y 443.136,Z 749.56,A -85,B 0,C 180,E1 15288.188,E2 15288.188} C_VEL
LIN {X 0,Y 443.536,Z 749.56,A -85,B 0,C 180,E1 15294.128,E2 15294.128} C_VEL
LIN {X 0,Y 443.985,Z 749.56,A -85,B 0,C 180,E1 15299.995,E2 15299.995} C_VEL
LIN {X 0,Y 443.589,Z 749.56,A -85,B 0,C 180,E1 15305.86,E2 15305.86} C_VEL
LIN {X 0,Y 443.203,Z 749.56,A -85,B 0,C 180,E1 15311.799,E2 15311.799} C_VEL
LIN {X 0,Y 442.969,Z 749.848,A -85,B 0,C 180,E1 15316.461,E2 15316.461} C_VEL
LIN {X 0,Y 444.959,Z 754.776,A -85,B 0,C 180,E1 15317.257,E2 15317.257} C_VEL
LIN {X 0,Y 448.517,Z 758.374,A -85,B 0,C 180,E1 15318.408,E2 15318.408} C_VEL
LIN {X 0,Y 455.021,Z 767.666,A -85,B 0,C 180,E1 15320.449,E2 15320.449} C_VEL
LIN {X 0,Y 467.929,Z 785.183,A -85,B 0,C 180,E1 15323.969,E2 15323.969} C_VEL
LIN {X 0,Y 487.495,Z 814.955,A -85,B 0,C 180,E1 15328.553,E2 15328.553} C_VEL
LIN {X 0,Y 506.44,Z 848.845,A -85,B 0,C 180,E1 15332.689,E2 15332.689} C_VEL
LIN {X 0,Y 521.542,Z 881.372,A -85,B 0,C 180,E1 15336.141,E2 15336.141} C_VEL
LIN {X 0,Y 513.713,Z 926.44,A -85,B 0,C 180,E1 15337.81,E2 15337.81} C_VEL
LIN {X 0,Y 503.664,Z 972.981,A -85,B 0,C 180,E1 15340.292,E2 15340.292} C_VEL
LIN {X 0,Y 493.089,Z 1014.897,A -85,B 0,C 180,E1 15343.276,E2 15343.276} C_VEL
LIN {X 0,Y 481.25,Z 1056.049,A -85,B 0,C 180,E1 15347.129,E2 15347.129} C_VEL
LIN {X 0,Y 470.53,Z 1092.312,A -85,B 0,C 180,E1 15351.535,E2 15351.535} C_VEL
LIN {X 0,Y 460.291,Z 1126.735,A -85,B 0,C 180,E1 15356.988,E2 15356.988} C_VEL
LIN {X 0,Y 453.076,Z 1153.137,A -85,B 0,C 180,E1 15362.433,E2 15362.433} C_VEL
LIN {X 0,Y 448.264,Z 1174.593,A -85,B 0,C 180,E1 15368.233,E2 15368.233} C_VEL
LIN {X 0,Y 445.405,Z 1191.139,A -85,B 0,C 180,E1 15374.25,E2 15374.25} C_VEL
LIN {X 0,Y 444.209,Z 1202.027,A -85,B 0,C 180,E1 15380.206,E2 15380.206} C_VEL
LIN {X 0,Y 443.909,Z 1206.461,A -85,B 0,C 180,E1 15384.138,E2 15384.138} C_VEL
LIN {X 0,Y 443.981,Z 1209.029,A -85,B 0,C 180,E1 15389.999,E2 15389.999} C_VEL
LIN {X 0,Y 443.895,Z 1207.804,A -85,B 0,C 180,E1 15393.903,E2 15393.903} C_VEL
LIN {X 0,Y 444.075,Z 1204.368,A -85,B 0,C 180,E1 15397.987,E2 15397.987} C_VEL
LIN {X 0,Y 441.691,Z 1202.1,A -85,B 0,C 180,E1 15399.63,E2 15399.63} C_VEL
LIN {X 0,Y 436.67,Z 1198.023,A -85,B 0,C 180,E1 15402.087,E2 15402.087} C_VEL
LIN {X 0,Y 436.622,Z 1197.543,A -85,B 0,C 180,E1 15402.37,E2 15402.37} C_VEL
LIN {X 0,Y 438.6,Z 1184.251,A -85,B 0,C 180,E1 15408.537,E2 15408.537} C_VEL
LIN {X 0,Y 442.694,Z 1164.341,A -85,B 0,C 180,E1 15414.89,E2 15414.89} C_VEL
LIN {X 0,Y 449.476,Z 1138.715,A -85,B 0,C 180,E1 15421.036,E2 15421.036} C_VEL
LIN {X 0,Y 459.23,Z 1106.631,A -85,B 0,C 180,E1 15426.885,E2 15426.885} C_VEL
LIN {X 0,Y 470.535,Z 1071.818,A -85,B 0,C 180,E1 15431.788,E2 15431.788} C_VEL
LIN {X 0,Y 483.76,Z 1030.909,A -85,B 0,C 180,E1 15436.214,E2 15436.214} C_VEL
LIN {X 0,Y 496.587,Z 987.757,A -85,B 0,C 180,E1 15439.732,E2 15439.732} C_VEL
LIN {X 0,Y 508.604,Z 942.289,A -85,B 0,C 180,E1 15442.484,E2 15442.484} C_VEL
LIN {X 0,Y 518.066,Z 897.943,A -85,B 0,C 180,E1 15444.407,E2 15444.407} C_VEL
LIN {X 0,Y 520.031,Z 884.311,A -85,B 0,C 180,E1 15444.969,E2 15444.969} C_VEL
LIN {X 0,Y 510.451,Z 859.29,A -85,B 0,C 180,E1 15447.993,E2 15447.993} C_VEL
LIN {X 0,Y 497.648,Z 834.956,A -85,B 0,C 180,E1 15451.829,E2 15451.829} C_VEL
LIN {X 0,Y 483.858,Z 813.022,A -85,B 0,C 180,E1 15456.376,E2 15456.376} C_VEL
LIN {X 0,Y 474.386,Z 799.72,A -85,B 0,C 180,E1 15460.101,E2 15460.101} C_VEL
LIN {X 0,Y 469.701,Z 793.316,A -85,B 0,C 180,E1 15462.269,E2 15462.269} C_VEL
LIN {X 0,Y 465.275,Z 787.037,A -85,B 0,C 180,E1 15464.704,E2 15464.704} C_VEL
LIN {X 0,Y 460.36,Z 780.143,A -85,B 0,C 180,E1 15468.166,E2 15468.166} C_VEL
LIN {X 0,Y 456.125,Z 774.273,A -85,B 0,C 180,E1 15472.928,E2 15472.928} C_VEL
LIN {X 0,Y 455.48,Z 772.875,A -85,B 0,C 180,E1 15474.293,E2 15474.293} C_VEL
LIN {X 0,Y 456.293,Z 773.673,A -85,B 0,C 180,E1 15482.675,E2 15482.675} C_VEL
LIN {X 0,Y 459.504,Z 779.493,A -85,B 0,C 180,E1 15486.615,E2 15486.615} C_VEL
LIN {X 0,Y 461.772,Z 781.669,A -85,B 0,C 180,E1 15488.394,E2 15488.394} C_VEL
LIN {X 0,Y 466.316,Z 787.595,A -85,B 0,C 180,E1 15491.335,E2 15491.335} C_VEL
LIN {X 0,Y 473.077,Z 798.068,A -85,B 0,C 180,E1 15494.93,E2 15494.93} C_VEL
LIN {X 0,Y 481.266,Z 809.796,A -85,B 0,C 180,E1 15498.424,E2 15498.424} C_VEL
LIN {X 0,Y 494.332,Z 831.4,A -85,B 0,C 180,E1 15503.287,E2 15503.287} C_VEL
LIN {X 0,Y 507.111,Z 857.373,A -85,B 0,C 180,E1 15507.755,E2 15507.755} C_VEL
LIN {X 0,Y 515.093,Z 878.982,A -85,B 0,C 180,E1 15510.806,E2 15510.806} C_VEL
LIN {X 0,Y 504.938,Z 922.869,A -85,B 0,C 180,E1 15513.077,E2 15513.077} C_VEL
LIN {X 0,Y 492.547,Z 964.937,A -85,B 0,C 180,E1 15516.079,E2 15516.079} C_VEL
LIN {X 0,Y 480.067,Z 1001.966,A -85,B 0,C 180,E1 15519.638,E2 15519.638} C_VEL
LIN {X 0,Y 466.924,Z 1037.875,A -85,B 0,C 180,E1 15524.254,E2 15524.254} C_VEL
LIN {X 0,Y 455.387,Z 1068.669,A -85,B 0,C 180,E1 15529.634,E2 15529.634} C_VEL
LIN {X 0,Y 447.223,Z 1091.494,A -85,B 0,C 180,E1 15534.943,E2 15534.943} C_VEL
LIN {X 0,Y 441.007,Z 1111.711,A -85,B 0,C 180,E1 15541.334,E2 15541.334} C_VEL
LIN {X 0,Y 437.788,Z 1125.298,A -85,B 0,C 180,E1 15547.687,E2 15547.687} C_VEL
LIN {X 0,Y 436.533,Z 1132.493,A -85,B 0,C 180,E1 15552.958,E2 15552.958} C_VEL
LIN {X 0,Y 435.958,Z 1135.978,A -85,B 0,C 180,E1 15557.997,E2 15557.997} C_VEL
LIN {X 0,Y 436.087,Z 1135.782,A -85,B 0,C 180,E1 15564.034,E2 15564.034} C_VEL
LIN {X 0,Y 436.869,Z 1130.936,A -85,B 0,C 180,E1 15570.001,E2 15570.001} C_VEL
LIN {X 0,Y 438.357,Z 1121.44,A -85,B 0,C 180,E1 15575.937,E2 15575.937} C_VEL
LIN {X 0,Y 441.642,Z 1106.802,A -85,B 0,C 180,E1 15581.848,E2 15581.848} C_VEL
LIN {X 0,Y 447.568,Z 1086.508,A -85,B 0,C 180,E1 15587.691,E2 15587.691} C_VEL
LIN {X 0,Y 456.613,Z 1059.436,A -85,B 0,C 180,E1 15593.4,E2 15593.4} C_VEL
LIN {X 0,Y 467.533,Z 1026.871,A -85,B 0,C 180,E1 15598.474,E2 15598.474} C_VEL
LIN {X 0,Y 478.613,Z 992.861,A -85,B 0,C 180,E1 15602.463,E2 15602.463} C_VEL
LIN {X 0,Y 490.257,Z 953.33,A -85,B 0,C 180,E1 15605.986,E2 15605.986} C_VEL
LIN {X 0,Y 501.173,Z 909.071,A -85,B 0,C 180,E1 15608.869,E2 15608.869} C_VEL
LIN {X 0,Y 507.811,Z 876.905,A -85,B 0,C 180,E1 15610.422,E2 15610.422} C_VEL
LIN {X 0,Y 493.822,Z 842.854,A -85,B 0,C 180,E1 15614.536,E2 15614.536} C_VEL
LIN {X 0,Y 477.866,Z 812.662,A -85,B 0,C 180,E1 15618.762,E2 15618.762} C_VEL
LIN {X 0,Y 459.681,Z 784.364,A -85,B 0,C 180,E1 15623.638,E2 15623.638} C_VEL
LIN {X 0,Y 448.287,Z 769.726,A -85,B 0,C 180,E1 15626.995,E2 15626.995} C_VEL
LIN {X 0,Y 443.711,Z 763.479,A -85,B 0,C 180,E1 15628.525,E2 15628.525} C_VEL
LIN {X 0,Y 439.842,Z 757.597,A -85,B 0,C 180,E1 15629.947,E2 15629.947} C_VEL
LIN {X 0,Y 434.857,Z 752.306,A -85,B 0,C 180,E1 15631.845,E2 15631.845} C_VEL
LIN {X 0,Y 434.35,Z 749.56,A -85,B 0,C 180,E1 15632.251,E2 15632.251} C_VEL
LIN {X 0,Y 434.52,Z 749.56,A -85,B 0,C 180,E1 15637.502,E2 15637.502} C_VEL
LIN {X 0,Y 434.851,Z 749.56,A -85,B 0,C 180,E1 15643.853,E2 15643.853} C_VEL
LIN {X 0,Y 435.365,Z 749.56,A -85,B 0,C 180,E1 15650,E2 15650} C_VEL
LIN {X 0,Y 435.826,Z 749.56,A -85,B 0,C 180,E1 15656.018,E2 15656.018} C_VEL
LIN {X 0,Y 435.949,Z 749.56,A -85,B 0,C 180,E1 15661.981,E2 15661.981} C_VEL
LIN {X 0,Y 435.523,Z 749.56,A -85,B 0,C 180,E1 15667.972,E2 15667.972} C_VEL
LIN {X 0,Y 435.237,Z 749.976,A -85,B 0,C 180,E1 15673.935,E2 15673.935} C_VEL
LIN {X 0,Y 437.183,Z 754.897,A -85,B 0,C 180,E1 15674.828,E2 15674.828} C_VEL
LIN {X 0,Y 440.813,Z 758.353,A -85,B 0,C 180,E1 15676.149,E2 15676.149} C_VEL
LIN {X 0,Y 445.19,Z 763.968,A -85,B 0,C 180,E1 15677.685,E2 15677.685} C_VEL
LIN {X 0,Y 461.256,Z 786.494,A -85,B 0,C 180,E1 15682.555,E2 15682.555} C_VEL
LIN {X 0,Y 478.398,Z 812.022,A -85,B 0,C 180,E1 15686.845,E2 15686.845} C_VEL
LIN {X 0,Y 497.582,Z 845.42,A -85,B 0,C 180,E1 15691.245,E2 15691.245} C_VEL
LIN {X 0,Y 515.839,Z 884.192,A -85,B 0,C 180,E1 15695.567,E2 15695.567} C_VEL
LIN {X 0,Y 507.491,Z 929.838,A -85,B 0,C 180,E1 15697.324,E2 15697.324} C_VEL
LIN {X 0,Y 496.862,Z 977.26,A -85,B 0,C 180,E1 15699.927,E2 15699.927} C_VEL
LIN {X 0,Y 485.962,Z 1018.084,A -85,B 0,C 180,E1 15702.94,E2 15702.94} C_VEL
LIN {X 0,Y 473.987,Z 1058.579,A -85,B 0,C 180,E1 15706.838,E2 15706.838} C_VEL
LIN {X 0,Y 462.867,Z 1094.587,A -85,B 0,C 180,E1 15711.362,E2 15711.362} C_VEL
LIN {X 0,Y 452.722,Z 1127.706,A -85,B 0,C 180,E1 15716.744,E2 15716.744} C_VEL
LIN {X 0,Y 445.089,Z 1154.552,A -85,B 0,C 180,E1 15722.475,E2 15722.475} C_VEL
LIN {X 0,Y 440.274,Z 1175.51,A -85,B 0,C 180,E1 15728.347,E2 15728.347} C_VEL
LIN {X 0,Y 437.596,Z 1190.456,A -85,B 0,C 180,E1 15733.962,E2 15733.962} C_VEL
LIN {X 0,Y 436.334,Z 1201.37,A -85,B 0,C 180,E1 15740.027,E2 15740.027} C_VEL
LIN {X 0,Y 436.024,Z 1205.811,A -85,B 0,C 180,E1 15744.031,E2 15744.031} C_VEL
LIN {X 0,Y 436.124,Z 1208.382,A -85,B 0,C 180,E1 15749.999,E2 15749.999} C_VEL
LIN {X 0,Y 436.019,Z 1207.148,A -85,B 0,C 180,E1 15753.974,E2 15753.974} C_VEL
LIN {X 0,Y 436.282,Z 1203.041,A -85,B 0,C 180,E1 15758.649,E2 15758.649} C_VEL
LIN {X 0,Y 436.622,Z 1197.543,A -85,B 0,C 180,E1 15762.37,E2 15762.37} C_VEL
LIN {X 0,Y 433.159,Z 1193.433,A -85,B 0,C 180,E1 15764.569,E2 15764.569} C_VEL
LIN {X 0,Y 429.971,Z 1188.56,A -85,B 0,C 180,E1 15766.777,E2 15766.777} C_VEL
LIN {X 0,Y 433.259,Z 1171.232,A -85,B 0,C 180,E1 15773.102,E2 15773.102} C_VEL
LIN {X 0,Y 439.286,Z 1148.069,A -85,B 0,C 180,E1 15779.352,E2 15779.352} C_VEL
LIN {X 0,Y 448.863,Z 1116.968,A -85,B 0,C 180,E1 15785.682,E2 15785.682} C_VEL
LIN {X 0,Y 459.948,Z 1083.84,A -85,B 0,C 180,E1 15790.834,E2 15790.834} C_VEL
LIN {X 0,Y 473.361,Z 1044.613,A -85,B 0,C 180,E1 15795.539,E2 15795.539} C_VEL
LIN {X 0,Y 487.24,Z 1001.247,A -85,B 0,C 180,E1 15799.431,E2 15799.431} C_VEL
LIN {X 0,Y 499.53,Z 958.634,A -85,B 0,C 180,E1 15802.298,E2 15802.298} C_VEL
LIN {X 0,Y 509.784,Z 915.602,A -85,B 0,C 180,E1 15804.437,E2 15804.437} C_VEL
LIN {X 0,Y 514.996,Z 888.308,A -85,B 0,C 180,E1 15805.515,E2 15805.515} C_VEL
LIN {X 0,Y 506.209,Z 864.374,A -85,B 0,C 180,E1 15808.511,E2 15808.511} C_VEL
LIN {X 0,Y 493.517,Z 839.651,A -85,B 0,C 180,E1 15812.538,E2 15812.538} C_VEL
LIN {X 0,Y 480.853,Z 819.096,A -85,B 0,C 180,E1 15816.976,E2 15816.976} C_VEL
LIN {X 0,Y 472.19,Z 806.661,A -85,B 0,C 180,E1 15820.523,E2 15820.523} C_VEL
LIN {X 0,Y 467.813,Z 800.394,A -85,B 0,C 180,E1 15822.68,E2 15822.68} C_VEL
LIN {X 0,Y 463.927,Z 794.669,A -85,B 0,C 180,E1 15824.9,E2 15824.9} C_VEL
LIN {X 0,Y 459.105,Z 787.819,A -85,B 0,C 180,E1 15828.374,E2 15828.374} C_VEL
LIN {X 0,Y 455.007,Z 781.745,A -85,B 0,C 180,E1 15833.21,E2 15833.21} C_VEL
LIN {X 0,Y 453.871,Z 780.511,A -85,B 0,C 180,E1 15836.187,E2 15836.187} C_VEL
LIN {X 0,Y 455.24,Z 781.546,A -85,B 0,C 180,E1 15842.562,E2 15842.562} C_VEL
LIN {X 0,Y 458.543,Z 787.359,A -85,B 0,C 180,E1 15846.629,E2 15846.629} C_VEL
LIN {X 0,Y 460.547,Z 789.534,A -85,B 0,C 180,E1 15848.242,E2 15848.242} C_VEL
LIN {X 0,Y 465.745,Z 797.31,A -85,B 0,C 180,E1 15851.765,E2 15851.765} C_VEL
LIN {X 0,Y 471.627,Z 806.048,A -85,B 0,C 180,E1 15854.858,E2 15854.858} C_VEL
LIN {X 0,Y 480.51,Z 819.601,A -85,B 0,C 180,E1 15858.811,E2 15858.811} C_VEL
LIN {X 0,Y 492.598,Z 840.958,A -85,B 0,C 180,E1 15863.509,E2 15863.509} C_VEL
LIN {X 0,Y 503.787,Z 865.305,A -85,B 0,C 180,E1 15867.712,E2 15867.712} C_VEL
LIN {X 0,Y 509.933,Z 883.171,A -85,B 0,C 180,E1 15870.256,E2 15870.256} C_VEL
LIN {X 0,Y 499.768,Z 924.654,A -85,B 0,C 180,E1 15872.427,E2 15872.427} C_VEL
LIN {X 0,Y 486.713,Z 967.519,A -85,B 0,C 180,E1 15875.527,E2 15875.527} C_VEL
LIN {X 0,Y 473.702,Z 1004.482,A -85,B 0,C 180,E1 15879.157,E2 15879.157} C_VEL
LIN {X 0,Y 461.033,Z 1037.875,A -85,B 0,C 180,E1 15883.505,E2 15883.505} C_VEL
LIN {X 0,Y 449.134,Z 1068.135,A -85,B 0,C 180,E1 15888.799,E2 15888.799} C_VEL
LIN {X 0,Y 440.227,Z 1091.735,A -85,B 0,C 180,E1 15894.301,E2 15894.301} C_VEL
LIN {X 0,Y 433.588,Z 1112.039,A -85,B 0,C 180,E1 15900.797,E2 15900.797} C_VEL
LIN {X 0,Y 430.095,Z 1125.734,A -85,B 0,C 180,E1 15907.265,E2 15907.265} C_VEL
LIN {X 0,Y 428.797,Z 1132.43,A -85,B 0,C 180,E1 15912.106,E2 15912.106} C_VEL
LIN {X 0,Y 428.076,Z 1136.568,A -85,B 0,C 180,E1 15917.773,E2 15917.773} C_VEL
LIN {X 0,Y 428.218,Z 1136.498,A -85,B 0,C 180,E1 15923.924,E2 15923.924} C_VEL
LIN {X 0,Y 428.765,Z 1132.878,A -85,B 0,C 180,E1 15928.991,E2 15928.991} C_VEL
LIN {X 0,Y 430.28,Z 1124.227,A -85,B 0,C 180,E1 15935.038,E2 15935.038} C_VEL
LIN {X 0,Y 433.306,Z 1110.677,A -85,B 0,C 180,E1 15941.059,E2 15941.059} C_VEL
LIN {X 0,Y 439.515,Z 1089.689,A -85,B 0,C 180,E1 15947.509,E2 15947.509} C_VEL
LIN {X 0,Y 448.144,Z 1064.477,A -85,B 0,C 180,E1 15953.08,E2 15953.08} C_VEL
LIN {X 0,Y 458.58,Z 1034.939,A -85,B 0,C 180,E1 15958.008,E2 15958.008} C_VEL
LIN {X 0,Y 470.826,Z 998.91,A -85,B 0,C 180,E1 15962.521,E2 15962.521} C_VEL
LIN {X 0,Y 482.511,Z 960.635,A -85,B 0,C 180,E1 15966.099,E2 15966.099} C_VEL
LIN {X 0,Y 493.623,Z 918.858,A -85,B 0,C 180,E1 15969.013,E2 15969.013} C_VEL
LIN {X 0,Y 502.012,Z 879.714,A -85,B 0,C 180,E1 15971.017,E2 15971.017} C_VEL
LIN {X 0,Y 487.066,Z 843.536,A -85,B 0,C 180,E1 15975.579,E2 15975.579} C_VEL
LIN {X 0,Y 471.526,Z 814.093,A -85,B 0,C 180,E1 15979.91,E2 15979.91} C_VEL
LIN {X 0,Y 455.5,Z 789.506,A -85,B 0,C 180,E1 15984.425,E2 15984.425} C_VEL
LIN {X 0,Y 444.668,Z 775.068,A -85,B 0,C 180,E1 15987.799,E2 15987.799} C_VEL
LIN {X 0,Y 440.651,Z 769.841,A -85,B 0,C 180,E1 15989.188,E2 15989.188} C_VEL
LIN {X 0,Y 436.331,Z 763.763,A -85,B 0,C 180,E1 15990.823,E2 15990.823} C_VEL
LIN {X 0,Y 432.343,Z 758.087,A -85,B 0,C 180,E1 15992.478,E2 15992.478} C_VEL
LIN {X 0,Y 426.899,Z 752.052,A -85,B 0,C 180,E1 15994.927,E2 15994.927} C_VEL
LIN {X 0,Y 426.538,Z 749.56,A -85,B 0,C 180,E1 15995.394,E2 15995.394} C_VEL
LIN {X 0,Y 426.761,Z 749.56,A -85,B 0,C 180,E1 16001.41,E2 16001.41} C_VEL
LIN {X 0,Y 427.271,Z 749.56,A -85,B 0,C 180,E1 16007.743,E2 16007.743} C_VEL
LIN {X 0,Y 427.702,Z 749.56,A -85,B 0,C 180,E1 16013.91,E2 16013.91} C_VEL
LIN {X 0,Y 428.192,Z 749.56,A -85,B 0,C 180,E1 16019.994,E2 16019.994} C_VEL
LIN {X 0,Y 427.747,Z 749.56,A -85,B 0,C 180,E1 16026.078,E2 16026.078} C_VEL
LIN {X 0,Y 427.425,Z 750.311,A -85,B 0,C 180,E1 16030.949,E2 16030.949} C_VEL
LIN {X 0,Y 429.655,Z 755.106,A -85,B 0,C 180,E1 16032.113,E2 16032.113} C_VEL
LIN {X 0,Y 433.155,Z 758.083,A -85,B 0,C 180,E1 16033.575,E2 16033.575} C_VEL
LIN {X 0,Y 436.872,Z 763.62,A -85,B 0,C 180,E1 16035.111,E2 16035.111} C_VEL
LIN {X 0,Y 438.924,Z 766.209,A -85,B 0,C 180,E1 16035.886,E2 16035.886} C_VEL
LIN {X 0,Y 445.281,Z 774.923,A -85,B 0,C 180,E1 16038.134,E2 16038.134} C_VEL
LIN {X 0,Y 457.998,Z 792.248,A -85,B 0,C 180,E1 16041.993,E2 16041.993} C_VEL
LIN {X 0,Y 476.699,Z 820.782,A -85,B 0,C 180,E1 16046.814,E2 16046.814} C_VEL
LIN {X 0,Y 495.105,Z 854.776,A -85,B 0,C 180,E1 16051.293,E2 16051.293} C_VEL
LIN {X 0,Y 510.014,Z 888.003,A -85,B 0,C 180,E1 16055.024,E2 16055.024} C_VEL
LIN {X 0,Y 500.958,Z 934.804,A -85,B 0,C 180,E1 16056.9,E2 16056.9} C_VEL
LIN {X 0,Y 490.296,Z 980.306,A -85,B 0,C 180,E1 16059.481,E2 16059.481} C_VEL
LIN {X 0,Y 478.074,Z 1023.97,A -85,B 0,C 180,E1 16062.831,E2 16062.831} C_VEL
LIN {X 0,Y 466.466,Z 1061.817,A -85,B 0,C 180,E1 16066.62,E2 16066.62} C_VEL
LIN {X 0,Y 454.281,Z 1099.683,A -85,B 0,C 180,E1 16071.599,E2 16071.599} C_VEL
LIN {X 0,Y 444.666,Z 1129.99,A -85,B 0,C 180,E1 16076.764,E2 16076.764} C_VEL
LIN {X 0,Y 436.872,Z 1156.941,A -85,B 0,C 180,E1 16082.77,E2 16082.77} C_VEL
LIN {X 0,Y 432.257,Z 1176.57,A -85,B 0,C 180,E1 16088.512,E2 16088.512} C_VEL
LIN {X 0,Y 429.568,Z 1191.29,A -85,B 0,C 180,E1 16094.394,E2 16094.394} C_VEL
LIN {X 0,Y 428.486,Z 1200.713,A -85,B 0,C 180,E1 16099.843,E2 16099.843} C_VEL
LIN {X 0,Y 428.139,Z 1205.159,A -85,B 0,C 180,E1 16103.921,E2 16103.921} C_VEL
LIN {X 0,Y 428.248,Z 1207.734,A -85,B 0,C 180,E1 16109.999,E2 16109.999} C_VEL
LIN {X 0,Y 428.132,Z 1206.492,A -85,B 0,C 180,E1 16114.047,E2 16114.047} C_VEL
LIN {X 0,Y 428.386,Z 1202.091,A -85,B 0,C 180,E1 16119.023,E2 16119.023} C_VEL
LIN {X 0,Y 429.354,Z 1192.624,A -85,B 0,C 180,E1 16124.867,E2 16124.867} C_VEL
LIN {X 0,Y 429.971,Z 1188.56,A -85,B 0,C 180,E1 16126.777,E2 16126.777} C_VEL
LIN {X 0,Y 429.179,Z 1185.973,A -85,B 0,C 180,E1 16127.884,E2 16127.884} C_VEL
LIN {X 0,Y 424.05,Z 1178.291,A -85,B 0,C 180,E1 16130.906,E2 16130.906} C_VEL
LIN {X 0,Y 424.12,Z 1177.532,A -85,B 0,C 180,E1 16131.186,E2 16131.186} C_VEL
LIN {X 0,Y 428.936,Z 1157.857,A -85,B 0,C 180,E1 16137.256,E2 16137.256} C_VEL
LIN {X 0,Y 437.272,Z 1130.683,A -85,B 0,C 180,E1 16143.567,E2 16143.567} C_VEL
LIN {X 0,Y 447.934,Z 1099.628,A -85,B 0,C 180,E1 16149.119,E2 16149.119} C_VEL
LIN {X 0,Y 461.639,Z 1061.13,A -85,B 0,C 180,E1 16154.367,E2 16154.367} C_VEL
LIN {X 0,Y 475.143,Z 1021.91,A -85,B 0,C 180,E1 16158.407,E2 16158.407} C_VEL
LIN {X 0,Y 488.934,Z 978.122,A -85,B 0,C 180,E1 16161.825,E2 16161.825} C_VEL
LIN {X 0,Y 501.304,Z 931.517,A -85,B 0,C 180,E1 16164.476,E2 16164.476} C_VEL
LIN {X 0,Y 509.981,Z 892.396,A -85,B 0,C 180,E1 16166.063,E2 16166.063} C_VEL
LIN {X 0,Y 501.894,Z 869.452,A -85,B 0,C 180,E1 16169.007,E2 16169.007} C_VEL
LIN {X 0,Y 489.562,Z 844.591,A -85,B 0,C 180,E1 16173.197,E2 16173.197} C_VEL
LIN {X 0,Y 476.221,Z 822.208,A -85,B 0,C 180,E1 16178.246,E2 16178.246} C_VEL
LIN {X 0,Y 466.375,Z 808.196,A -85,B 0,C 180,E1 16182.79,E2 16182.79} C_VEL
LIN {X 0,Y 462.304,Z 802.168,A -85,B 0,C 180,E1 16185.21,E2 16185.21} C_VEL
LIN {X 0,Y 457.852,Z 795.537,A -85,B 0,C 180,E1 16188.583,E2 16188.583} C_VEL
LIN {X 0,Y 453.9,Z 789.222,A -85,B 0,C 180,E1 16193.494,E2 16193.494} C_VEL
LIN {X 0,Y 454.081,Z 788.715,A -85,B 0,C 180,E1 16202.151,E2 16202.151} C_VEL
LIN {X 0,Y 456.933,Z 794.815,A -85,B 0,C 180,E1 16206.176,E2 16206.176} C_VEL
LIN {X 0,Y 459.16,Z 797.34,A -85,B 0,C 180,E1 16208.093,E2 16208.093} C_VEL
LIN {X 0,Y 464.369,Z 805.287,A -85,B 0,C 180,E1 16211.681,E2 16211.681} C_VEL
LIN {X 0,Y 471.98,Z 816.719,A -85,B 0,C 180,E1 16215.797,E2 16215.797} C_VEL
LIN {X 0,Y 483.067,Z 835.802,A -85,B 0,C 180,E1 16220.717,E2 16220.717} C_VEL
LIN {X 0,Y 494.613,Z 859.083,A -85,B 0,C 180,E1 16225.329,E2 16225.329} C_VEL
LIN {X 0,Y 504.214,Z 884.691,A -85,B 0,C 180,E1 16229.363,E2 16229.363} C_VEL
LIN {X 0,Y 504.549,Z 888.16,A -85,B 0,C 180,E1 16229.711,E2 16229.711} C_VEL
LIN {X 0,Y 493.826,Z 929.363,A -85,B 0,C 180,E1 16231.955,E2 16231.955} C_VEL
LIN {X 0,Y 480.762,Z 970.575,A -85,B 0,C 180,E1 16234.999,E2 16234.999} C_VEL
LIN {X 0,Y 466.987,Z 1008.032,A -85,B 0,C 180,E1 16238.782,E2 16238.782} C_VEL
LIN {X 0,Y 453.779,Z 1041.22,A -85,B 0,C 180,E1 16243.244,E2 16243.244} C_VEL
LIN {X 0,Y 441.707,Z 1070.912,A -85,B 0,C 180,E1 16248.611,E2 16248.611} C_VEL
LIN {X 0,Y 432.299,Z 1094.717,A -85,B 0,C 180,E1 16254.425,E2 16254.425} C_VEL
LIN {X 0,Y 425.78,Z 1113.743,A -85,B 0,C 180,E1 16260.792,E2 16260.792} C_VEL
LIN {X 0,Y 422.442,Z 1126.174,A -85,B 0,C 180,E1 16266.83,E2 16266.83} C_VEL
LIN {X 0,Y 420.727,Z 1134.536,A -85,B 0,C 180,E1 16273.303,E2 16273.303} C_VEL
LIN {X 0,Y 420.142,Z 1137.676,A -85,B 0,C 180,E1 16279.641,E2 16279.641} C_VEL
LIN {X 0,Y 420.631,Z 1136.217,A -85,B 0,C 180,E1 16285.881,E2 16285.881} C_VEL
LIN {X 0,Y 421.507,Z 1129.978,A -85,B 0,C 180,E1 16292.056,E2 16292.056} C_VEL
LIN {X 0,Y 423.751,Z 1119.084,A -85,B 0,C 180,E1 16298.202,E2 16298.202} C_VEL
LIN {X 0,Y 428.195,Z 1102.882,A -85,B 0,C 180,E1 16304.303,E2 16304.303} C_VEL
LIN {X 0,Y 435.57,Z 1080.845,A -85,B 0,C 180,E1 16310.301,E2 16310.301} C_VEL
LIN {X 0,Y 445.788,Z 1052.766,A -85,B 0,C 180,E1 16315.867,E2 16315.867} C_VEL
LIN {X 0,Y 456.676,Z 1022.449,A -85,B 0,C 180,E1 16320.423,E2 16320.423} C_VEL
LIN {X 0,Y 469.335,Z 985.501,A -85,B 0,C 180,E1 16324.601,E2 16324.601} C_VEL
LIN {X 0,Y 480.807,Z 947.683,A -85,B 0,C 180,E1 16327.798,E2 16327.798} C_VEL
LIN {X 0,Y 491.712,Z 905.196,A -85,B 0,C 180,E1 16330.488,E2 16330.488} C_VEL
LIN {X 0,Y 496.296,Z 884.076,A -85,B 0,C 180,E1 16331.51,E2 16331.51} C_VEL
LIN {X 0,Y 484.184,Z 852.495,A -85,B 0,C 180,E1 16335.531,E2 16335.531} C_VEL
LIN {X 0,Y 469.907,Z 823.941,A -85,B 0,C 180,E1 16339.738,E2 16339.738} C_VEL
LIN {X 0,Y 454.038,Z 797.823,A -85,B 0,C 180,E1 16344.447,E2 16344.447} C_VEL
LIN {X 0,Y 439.41,Z 777.772,A -85,B 0,C 180,E1 16349.245,E2 16349.245} C_VEL
LIN {X 0,Y 433.837,Z 770.599,A -85,B 0,C 180,E1 16351.363,E2 16351.363} C_VEL
LIN {X 0,Y 429.234,Z 764.197,A -85,B 0,C 180,E1 16353.346,E2 16353.346} C_VEL
LIN {X 0,Y 424.986,Z 758.988,A -85,B 0,C 180,E1 16355.368,E2 16355.368} C_VEL
LIN {X 0,Y 424.233,Z 757.097,A -85,B 0,C 180,E1 16355.811,E2 16355.811} C_VEL
LIN {X 0,Y 419.391,Z 752.892,A -85,B 0,C 180,E1 16358.481,E2 16358.481} C_VEL
LIN {X 0,Y 418.73,Z 749.56,A -85,B 0,C 180,E1 16359.1,E2 16359.1} C_VEL
LIN {X 0,Y 419.117,Z 749.56,A -85,B 0,C 180,E1 16365.375,E2 16365.375} C_VEL
LIN {X 0,Y 419.702,Z 749.56,A -85,B 0,C 180,E1 16371.714,E2 16371.714} C_VEL
LIN {X 0,Y 420.119,Z 749.56,A -85,B 0,C 180,E1 16377.933,E2 16377.933} C_VEL
LIN {X 0,Y 419.913,Z 749.56,A -85,B 0,C 180,E1 16384.122,E2 16384.122} C_VEL
LIN {X 0,Y 419.735,Z 750.045,A -85,B 0,C 180,E1 16387.271,E2 16387.271} C_VEL
LIN {X 0,Y 421.783,Z 755.001,A -85,B 0,C 180,E1 16388.661,E2 16388.661} C_VEL
LIN {X 0,Y 425.595,Z 758.276,A -85,B 0,C 180,E1 16390.608,E2 16390.608} C_VEL
LIN {X 0,Y 429.37,Z 763.778,A -85,B 0,C 180,E1 16392.443,E2 16392.443} C_VEL
LIN {X 0,Y 431.459,Z 766.191,A -85,B 0,C 180,E1 16393.347,E2 16393.347} C_VEL
LIN {X 0,Y 437.933,Z 775.231,A -85,B 0,C 180,E1 16395.955,E2 16395.955} C_VEL
LIN {X 0,Y 443.468,Z 782.572,A -85,B 0,C 180,E1 16397.915,E2 16397.915} C_VEL
LIN {X 0,Y 456.787,Z 801.268,A -85,B 0,C 180,E1 16402.006,E2 16402.006} C_VEL
LIN {X 0,Y 473.702,Z 827.845,A -85,B 0,C 180,E1 16406.521,E2 16406.521} C_VEL
LIN {X 0,Y 491.05,Z 861.005,A -85,B 0,C 180,E1 16410.959,E2 16410.959} C_VEL
LIN {X 0,Y 504.262,Z 890.931,A -85,B 0,C 180,E1 16414.441,E2 16414.441} C_VEL
LIN {X 0,Y 494.432,Z 939.73,A -85,B 0,C 180,E1 16416.462,E2 16416.462} C_VEL
LIN {X 0,Y 483.284,Z 984.533,A -85,B 0,C 180,E1 16419.11,E2 16419.11} C_VEL
LIN {X 0,Y 470.715,Z 1028.182,A -85,B 0,C 180,E1 16422.577,E2 16422.577} C_VEL
LIN {X 0,Y 458.489,Z 1066.07,A -85,B 0,C 180,E1 16426.547,E2 16426.547} C_VEL
LIN {X 0,Y 446.169,Z 1103.113,A -85,B 0,C 180,E1 16431.598,E2 16431.598} C_VEL
LIN {X 0,Y 435.951,Z 1134.227,A -85,B 0,C 180,E1 16437.206,E2 16437.206} C_VEL
LIN {X 0,Y 428.649,Z 1159.237,A -85,B 0,C 180,E1 16443.058,E2 16443.058} C_VEL
LIN {X 0,Y 423.69,Z 1180.041,A -85,B 0,C 180,E1 16449.65,E2 16449.65} C_VEL
LIN {X 0,Y 421.358,Z 1193.402,A -85,B 0,C 180,E1 16455.519,E2 16455.519} C_VEL
LIN {X 0,Y 420.475,Z 1202.648,A -85,B 0,C 180,E1 16461.734,E2 16461.734} C_VEL
LIN {X 0,Y 420.236,Z 1206.724,A -85,B 0,C 180,E1 16467.938,E2 16467.938} C_VEL
LIN {X 0,Y 420.435,Z 1206.723,A -85,B 0,C 180,E1 16472.059,E2 16472.059} C_VEL
LIN {X 0,Y 420.466,Z 1202.575,A -85,B 0,C 180,E1 16478.264,E2 16478.264} C_VEL
LIN {X 0,Y 421.373,Z 1193.129,A -85,B 0,C 180,E1 16484.538,E2 16484.538} C_VEL
LIN {X 0,Y 423.947,Z 1178.357,A -85,B 0,C 180,E1 16490.881,E2 16490.881} C_VEL
LIN {X 0,Y 424.12,Z 1177.532,A -85,B 0,C 180,E1 16491.186,E2 16491.186} C_VEL
LIN {X 0,Y 421.612,Z 1171.487,A -85,B 0,C 180,E1 16493.391,E2 16493.391} C_VEL
LIN {X 0,Y 419.531,Z 1164.756,A -85,B 0,C 180,E1 16495.584,E2 16495.584} C_VEL
LIN {X 0,Y 427.352,Z 1138.763,A -85,B 0,C 180,E1 16502.331,E2 16502.331} C_VEL
LIN {X 0,Y 437.858,Z 1108.819,A -85,B 0,C 180,E1 16508.188,E2 16508.188} C_VEL
LIN {X 0,Y 451.146,Z 1073.067,A -85,B 0,C 180,E1 16513.56,E2 16513.56} C_VEL
LIN {X 0,Y 465.756,Z 1032.891,A -85,B 0,C 180,E1 16518.089,E2 16518.089} C_VEL
LIN {X 0,Y 479.702,Z 991.338,A -85,B 0,C 180,E1 16521.638,E2 16521.638} C_VEL
LIN {X 0,Y 493.618,Z 943.772,A -85,B 0,C 180,E1 16524.6,E2 16524.6} C_VEL
LIN {X 0,Y 504.232,Z 899.139,A -85,B 0,C 180,E1 16526.572,E2 16526.572} C_VEL
LIN {X 0,Y 504.508,Z 894.23,A -85,B 0,C 180,E1 16526.868,E2 16526.868} C_VEL
LIN {X 0,Y 495.457,Z 869.574,A -85,B 0,C 180,E1 16530.285,E2 16530.285} C_VEL
LIN {X 0,Y 483.088,Z 845.21,A -85,B 0,C 180,E1 16534.784,E2 16534.784} C_VEL
LIN {X 0,Y 472.385,Z 827.401,A -85,B 0,C 180,E1 16539.165,E2 16539.165} C_VEL
LIN {X 0,Y 464.507,Z 815.419,A -85,B 0,C 180,E1 16543.134,E2 16543.134} C_VEL
LIN {X 0,Y 460.436,Z 809.436,A -85,B 0,C 180,E1 16545.634,E2 16545.634} C_VEL
LIN {X 0,Y 456.466,Z 803.228,A -85,B 0,C 180,E1 16548.79,E2 16548.79} C_VEL
LIN {X 0,Y 452.761,Z 796.719,A -85,B 0,C 180,E1 16553.778,E2 16553.778} C_VEL
LIN {X 0,Y 452.959,Z 796.855,A -85,B 0,C 180,E1 16562.156,E2 16562.156} C_VEL
LIN {X 0,Y 456.186,Z 802.958,A -85,B 0,C 180,E1 16566.545,E2 16566.545} C_VEL
LIN {X 0,Y 457.868,Z 805.383,A -85,B 0,C 180,E1 16568.028,E2 16568.028} C_VEL
LIN {X 0,Y 462.543,Z 812.842,A -85,B 0,C 180,E1 16571.489,E2 16571.489} C_VEL
LIN {X 0,Y 470.031,Z 824.624,A -85,B 0,C 180,E1 16575.685,E2 16575.685} C_VEL
LIN {X 0,Y 480.01,Z 842.516,A -85,B 0,C 180,E1 16580.387,E2 16580.387} C_VEL
LIN {X 0,Y 490.854,Z 865.634,A -85,B 0,C 180,E1 16585.049,E2 16585.049} C_VEL
LIN {X 0,Y 499.706,Z 890.497,A -85,B 0,C 180,E1 16589.025,E2 16589.025} C_VEL
LIN {X 0,Y 488.228,Z 932.986,A -85,B 0,C 180,E1 16591.398,E2 16591.398} C_VEL
LIN {X 0,Y 474.941,Z 973.171,A -85,B 0,C 180,E1 16594.429,E2 16594.429} C_VEL
LIN {X 0,Y 460.517,Z 1011.049,A -85,B 0,C 180,E1 16598.336,E2 16598.336} C_VEL
LIN {X 0,Y 446.864,Z 1043.837,A -85,B 0,C 180,E1 16602.872,E2 16602.872} C_VEL
LIN {X 0,Y 434.731,Z 1072.516,A -85,B 0,C 180,E1 16608.173,E2 16608.173} C_VEL
LIN {X 0,Y 424.948,Z 1096.072,A -85,B 0,C 180,E1 16614.076,E2 16614.076} C_VEL
LIN {X 0,Y 418.55,Z 1113.745,A -85,B 0,C 180,E1 16620.067,E2 16620.067} C_VEL
LIN {X 0,Y 414.788,Z 1126.621,A -85,B 0,C 180,E1 16626.376,E2 16626.376} C_VEL
LIN {X 0,Y 412.921,Z 1135.092,A -85,B 0,C 180,E1 16632.977,E2 16632.977} C_VEL
LIN {X 0,Y 412.266,Z 1138.309,A -85,B 0,C 180,E1 16639.441,E2 16639.441} C_VEL
LIN {X 0,Y 412.733,Z 1136.929,A -85,B 0,C 180,E1 16645.802,E2 16645.802} C_VEL
LIN {X 0,Y 413.665,Z 1130.822,A -85,B 0,C 180,E1 16652.095,E2 16652.095} C_VEL
LIN {X 0,Y 415.981,Z 1120.019,A -85,B 0,C 180,E1 16658.356,E2 16658.356} C_VEL
LIN {X 0,Y 420.609,Z 1103.972,A -85,B 0,C 180,E1 16664.567,E2 16664.567} C_VEL
LIN {X 0,Y 428.259,Z 1082.049,A -85,B 0,C 180,E1 16670.663,E2 16670.663} C_VEL
LIN {X 0,Y 438.621,Z 1054.566,A -85,B 0,C 180,E1 16676.236,E2 16676.236} C_VEL
LIN {X 0,Y 450.033,Z 1024.054,A -85,B 0,C 180,E1 16680.921,E2 16680.921} C_VEL
LIN {X 0,Y 463.279,Z 986.604,A -85,B 0,C 180,E1 16685.211,E2 16685.211} C_VEL
LIN {X 0,Y 475.029,Z 949.056,A -85,B 0,C 180,E1 16688.422,E2 16688.422} C_VEL
LIN {X 0,Y 486.366,Z 906.146,A -85,B 0,C 180,E1 16691.164,E2 16691.164} C_VEL
LIN {X 0,Y 490.696,Z 887.103,A -85,B 0,C 180,E1 16692.1,E2 16692.1} C_VEL
LIN {X 0,Y 477.108,Z 852.027,A -85,B 0,C 180,E1 16696.76,E2 16696.76} C_VEL
LIN {X 0,Y 462.778,Z 823.825,A -85,B 0,C 180,E1 16701.195,E2 16701.195} C_VEL
LIN {X 0,Y 447.282,Z 798.68,A -85,B 0,C 180,E1 16706.113,E2 16706.113} C_VEL
LIN {X 0,Y 432.543,Z 778.434,A -85,B 0,C 180,E1 16711.455,E2 16711.455} C_VEL
LIN {X 0,Y 426.966,Z 771.335,A -85,B 0,C 180,E1 16713.873,E2 16713.873} C_VEL
LIN {X 0,Y 422.891,Z 765.359,A -85,B 0,C 180,E1 16715.94,E2 16715.94} C_VEL
LIN {X 0,Y 417.588,Z 759.617,A -85,B 0,C 180,E1 16719.011,E2 16719.011} C_VEL
LIN {X 0,Y 416.771,Z 757.208,A -85,B 0,C 180,E1 16719.664,E2 16719.664} C_VEL
LIN {X 0,Y 411.784,Z 752.873,A -85,B 0,C 180,E1 16723.607,E2 16723.607} C_VEL
LIN {X 0,Y 411.146,Z 749.56,A -85,B 0,C 180,E1 16724.812,E2 16724.812} C_VEL
LIN {X 0,Y 411.778,Z 749.56,A -85,B 0,C 180,E1 16731.553,E2 16731.553} C_VEL
LIN {X 0,Y 412.209,Z 749.56,A -85,B 0,C 180,E1 16737.893,E2 16737.893} C_VEL
LIN {X 0,Y 412.22,Z 750.084,A -85,B 0,C 180,E1 16742.226,E2 16742.226} C_VEL
LIN {X 0,Y 413.807,Z 754.574,A -85,B 0,C 180,E1 16743.92,E2 16743.92} C_VEL
LIN {X 0,Y 418.192,Z 758.314,A -85,B 0,C 180,E1 16746.999,E2 16746.999} C_VEL
LIN {X 0,Y 421.656,Z 763.765,A -85,B 0,C 180,E1 16749.145,E2 16749.145} C_VEL
LIN {X 0,Y 423.94,Z 766.039,A -85,B 0,C 180,E1 16750.326,E2 16750.326} C_VEL
LIN {X 0,Y 428.402,Z 771.739,A -85,B 0,C 180,E1 16752.472,E2 16752.472} C_VEL
LIN {X 0,Y 440.297,Z 788.174,A -85,B 0,C 180,E1 16757.213,E2 16757.213} C_VEL
LIN {X 0,Y 454.331,Z 808.369,A -85,B 0,C 180,E1 16761.697,E2 16761.697} C_VEL
LIN {X 0,Y 470.387,Z 834.484,A -85,B 0,C 180,E1 16766.18,E2 16766.18} C_VEL
LIN {X 0,Y 487.036,Z 867.454,A -85,B 0,C 180,E1 16770.659,E2 16770.659} C_VEL
LIN {X 0,Y 498.446,Z 894.04,A -85,B 0,C 180,E1 16773.844,E2 16773.844} C_VEL
LIN {X 0,Y 488.382,Z 942.682,A -85,B 0,C 180,E1 16775.925,E2 16775.925} C_VEL
LIN {X 0,Y 476.195,Z 989.442,A -85,B 0,C 180,E1 16778.79,E2 16778.79} C_VEL
LIN {X 0,Y 463.774,Z 1030.562,A -85,B 0,C 180,E1 16782.159,E2 16782.159} C_VEL
LIN {X 0,Y 450.585,Z 1070.163,A -85,B 0,C 180,E1 16786.455,E2 16786.455} C_VEL
LIN {X 0,Y 438.729,Z 1104.394,A -85,B 0,C 180,E1 16791.295,E2 16791.295} C_VEL
LIN {X 0,Y 428.042,Z 1135.86,A -85,B 0,C 180,E1 16797.125,E2 16797.125} C_VEL
LIN {X 0,Y 421.014,Z 1159.088,A -85,B 0,C 180,E1 16802.733,E2 16802.733} C_VEL
LIN {X 0,Y 415.991,Z 1179.309,A -85,B 0,C 180,E1 16809.256,E2 16809.256} C_VEL
LIN {X 0,Y 413.403,Z 1193.748,A -85,B 0,C 180,E1 16815.771,E2 16815.771} C_VEL
LIN {X 0,Y 412.602,Z 1201.994,A -85,B 0,C 180,E1 16821.575,E2 16821.575} C_VEL
LIN {X 0,Y 412.355,Z 1206.076,A -85,B 0,C 180,E1 16827.899,E2 16827.899} C_VEL
LIN {X 0,Y 412.548,Z 1206.07,A -85,B 0,C 180,E1 16832.098,E2 16832.098} C_VEL
LIN {X 0,Y 412.589,Z 1201.719,A -85,B 0,C 180,E1 16838.579,E2 16838.579} C_VEL
LIN {X 0,Y 413.538,Z 1192.43,A -85,B 0,C 180,E1 16844.819,E2 16844.819} C_VEL
LIN {X 0,Y 416.286,Z 1177.668,A -85,B 0,C 180,E1 16851.284,E2 16851.284} C_VEL
LIN {X 0,Y 419.531,Z 1164.756,A -85,B 0,C 180,E1 16855.584,E2 16855.584} C_VEL
LIN {X 0,Y 419.346,Z 1161.244,A -85,B 0,C 180,E1 16856.672,E2 16856.672} C_VEL
LIN {X 0,Y 415.923,Z 1151.401,A -85,B 0,C 180,E1 16859.68,E2 16859.68} C_VEL
LIN {X 0,Y 416.16,Z 1150.403,A -85,B 0,C 180,E1 16859.949,E2 16859.949} C_VEL
LIN {X 0,Y 425.714,Z 1122.968,A -85,B 0,C 180,E1 16866.164,E2 16866.164} C_VEL
LIN {X 0,Y 439.028,Z 1088.162,A -85,B 0,C 180,E1 16872.13,E2 16872.13} C_VEL
LIN {X 0,Y 453.385,Z 1050.852,A -85,B 0,C 180,E1 16876.93,E2 16876.93} C_VEL
LIN {X 0,Y 468.444,Z 1009.829,A -85,B 0,C 180,E1 16880.929,E2 16880.929} C_VEL
LIN {X 0,Y 481.95,Z 968.188,A -85,B 0,C 180,E1 16883.945,E2 16883.945} C_VEL
LIN {X 0,Y 493.895,Z 924.785,A -85,B 0,C 180,E1 16886.291,E2 16886.291} C_VEL
LIN {X 0,Y 499.832,Z 898.992,A -85,B 0,C 180,E1 16887.358,E2 16887.358} C_VEL
LIN {X 0,Y 491.229,Z 874.797,A -85,B 0,C 180,E1 16890.812,E2 16890.812} C_VEL
LIN {X 0,Y 479.817,Z 851.506,A -85,B 0,C 180,E1 16895.217,E2 16895.217} C_VEL
LIN {X 0,Y 469.944,Z 834.378,A -85,B 0,C 180,E1 16899.518,E2 16899.518} C_VEL
LIN {X 0,Y 462.268,Z 822.339,A -85,B 0,C 180,E1 16903.59,E2 16903.59} C_VEL
LIN {X 0,Y 458.83,Z 816.914,A -85,B 0,C 180,E1 16905.906,E2 16905.906} C_VEL
LIN {X 0,Y 455.06,Z 810.903,A -85,B 0,C 180,E1 16908.997,E2 16908.997} C_VEL
LIN {X 0,Y 451.422,Z 804.13,A -85,B 0,C 180,E1 16914.242,E2 16914.242} C_VEL
LIN {X 0,Y 451.775,Z 804.945,A -85,B 0,C 180,E1 16922.162,E2 16922.162} C_VEL
LIN {X 0,Y 455.314,Z 810.971,A -85,B 0,C 180,E1 16926.872,E2 16926.872} C_VEL
LIN {X 0,Y 460.744,Z 820.557,A -85,B 0,C 180,E1 16931.355,E2 16931.355} C_VEL
LIN {X 0,Y 467.5,Z 831.775,A -85,B 0,C 180,E1 16935.412,E2 16935.412} C_VEL
LIN {X 0,Y 476.98,Z 849.668,A -85,B 0,C 180,E1 16940.159,E2 16940.159} C_VEL
LIN {X 0,Y 486.622,Z 871.143,A -85,B 0,C 180,E1 16944.564,E2 16944.564} C_VEL
LIN {X 0,Y 494.476,Z 894.065,A -85,B 0,C 180,E1 16948.375,E2 16948.375} C_VEL
LIN {X 0,Y 481.813,Z 939.476,A -85,B 0,C 180,E1 16951.014,E2 16951.014} C_VEL
LIN {X 0,Y 467.95,Z 978.913,A -85,B 0,C 180,E1 16954.137,E2 16954.137} C_VEL
LIN {X 0,Y 453.385,Z 1015.681,A -85,B 0,C 180,E1 16958.073,E2 16958.073} C_VEL
LIN {X 0,Y 438.497,Z 1049.926,A -85,B 0,C 180,E1 16963.063,E2 16963.063} C_VEL
LIN {X 0,Y 426.263,Z 1077.405,A -85,B 0,C 180,E1 16968.489,E2 16968.489} C_VEL
LIN {X 0,Y 416.574,Z 1100.156,A -85,B 0,C 180,E1 16974.522,E2 16974.522} C_VEL
LIN {X 0,Y 409.808,Z 1118.365,A -85,B 0,C 180,E1 16981.357,E2 16981.357} C_VEL
LIN {X 0,Y 406.297,Z 1130.503,A -85,B 0,C 180,E1 16988.167,E2 16988.167} C_VEL
LIN {X 0,Y 404.739,Z 1137.246,A -85,B 0,C 180,E1 16994.851,E2 16994.851} C_VEL
LIN {X 0,Y 404.451,Z 1139.037,A -85,B 0,C 180,E1 17001.406,E2 17001.406} C_VEL
LIN {X 0,Y 405.062,Z 1136.13,A -85,B 0,C 180,E1 17007.863,E2 17007.863} C_VEL
LIN {X 0,Y 406.002,Z 1130.218,A -85,B 0,C 180,E1 17013.202,E2 17013.202} C_VEL
LIN {X 0,Y 408.878,Z 1118.706,A -85,B 0,C 180,E1 17019.574,E2 17019.574} C_VEL
LIN {X 0,Y 414.743,Z 1100.219,A -85,B 0,C 180,E1 17026.403,E2 17026.403} C_VEL
LIN {X 0,Y 423.1,Z 1077.742,A -85,B 0,C 180,E1 17032.302,E2 17032.302} C_VEL
LIN {X 0,Y 434.089,Z 1049.934,A -85,B 0,C 180,E1 17037.75,E2 17037.75} C_VEL
LIN {X 0,Y 447.188,Z 1015.62,A -85,B 0,C 180,E1 17042.73,E2 17042.73} C_VEL
LIN {X 0,Y 460.101,Z 979,A -85,B 0,C 180,E1 17046.681,E2 17046.681} C_VEL
LIN {X 0,Y 473.021,Z 937.755,A -85,B 0,C 180,E1 17049.981,E2 17049.981} C_VEL
LIN {X 0,Y 484.278,Z 893.447,A -85,B 0,C 180,E1 17052.536,E2 17052.536} C_VEL
LIN {X 0,Y 484.648,Z 889.491,A -85,B 0,C 180,E1 17052.816,E2 17052.816} C_VEL
LIN {X 0,Y 471.881,Z 855.915,A -85,B 0,C 180,E1 17057.439,E2 17057.439} C_VEL
LIN {X 0,Y 457.762,Z 827.447,A -85,B 0,C 180,E1 17062.059,E2 17062.059} C_VEL
LIN {X 0,Y 443.715,Z 804.399,A -85,B 0,C 180,E1 17066.806,E2 17066.806} C_VEL
LIN {X 0,Y 430.649,Z 785.766,A -85,B 0,C 180,E1 17071.783,E2 17071.783} C_VEL
LIN {X 0,Y 424.86,Z 778.454,A -85,B 0,C 180,E1 17074.354,E2 17074.354} C_VEL
LIN {X 0,Y 420.168,Z 771.937,A -85,B 0,C 180,E1 17076.829,E2 17076.829} C_VEL
LIN {X 0,Y 415.933,Z 766.629,A -85,B 0,C 180,E1 17079.456,E2 17079.456} C_VEL
LIN {X 0,Y 414.793,Z 764.705,A -85,B 0,C 180,E1 17080.3,E2 17080.3} C_VEL
LIN {X 0,Y 410.309,Z 759.803,A -85,B 0,C 180,E1 17084.164,E2 17084.164} C_VEL
LIN {X 0,Y 409.739,Z 757.309,A -85,B 0,C 180,E1 17085.033,E2 17085.033} C_VEL
LIN {X 0,Y 406.429,Z 755.258,A -85,B 0,C 180,E1 17094.661,E2 17094.661} C_VEL
LIN {X 0,Y 410.916,Z 758.18,A -85,B 0,C 180,E1 17101.97,E2 17101.97} C_VEL
LIN {X 0,Y 413.637,Z 763.365,A -85,B 0,C 180,E1 17104.578,E2 17104.578} C_VEL
LIN {X 0,Y 416.688,Z 765.959,A -85,B 0,C 180,E1 17106.698,E2 17106.698} C_VEL
LIN {X 0,Y 420.715,Z 771.729,A -85,B 0,C 180,E1 17109.185,E2 17109.185} C_VEL
LIN {X 0,Y 422.687,Z 774.411,A -85,B 0,C 180,E1 17110.25,E2 17110.25} C_VEL
LIN {X 0,Y 428.269,Z 781.89,A -85,B 0,C 180,E1 17112.929,E2 17112.929} C_VEL
LIN {X 0,Y 438.287,Z 795.509,A -85,B 0,C 180,E1 17116.907,E2 17116.907} C_VEL
LIN {X 0,Y 453.345,Z 817.602,A -85,B 0,C 180,E1 17121.826,E2 17121.826} C_VEL
LIN {X 0,Y 469.845,Z 846.424,A -85,B 0,C 180,E1 17126.627,E2 17126.627} C_VEL
LIN {X 0,Y 484.892,Z 878.383,A -85,B 0,C 180,E1 17130.94,E2 17130.94} C_VEL
LIN {X 0,Y 492.686,Z 897.158,A -85,B 0,C 180,E1 17133.233,E2 17133.233} C_VEL
LIN {X 0,Y 482.49,Z 944.7,A -85,B 0,C 180,E1 17135.336,E2 17135.336} C_VEL
LIN {X 0,Y 469.484,Z 992.91,A -85,B 0,C 180,E1 17138.352,E2 17138.352} C_VEL
LIN {X 0,Y 455.968,Z 1035.573,A -85,B 0,C 180,E1 17142,E2 17142} C_VEL
LIN {X 0,Y 442.861,Z 1073.749,A -85,B 0,C 180,E1 17146.299,E2 17146.299} C_VEL
LIN {X 0,Y 430.036,Z 1109.3,A -85,B 0,C 180,E1 17151.599,E2 17151.599} C_VEL
LIN {X 0,Y 419.788,Z 1138.675,A -85,B 0,C 180,E1 17157.318,E2 17157.318} C_VEL
LIN {X 0,Y 412.027,Z 1163.963,A -85,B 0,C 180,E1 17163.888,E2 17163.888} C_VEL
LIN {X 0,Y 407.419,Z 1182.738,A -85,B 0,C 180,E1 17170.499,E2 17170.499} C_VEL
LIN {X 0,Y 405.167,Z 1195.589,A -85,B 0,C 180,E1 17177.068,E2 17177.068} C_VEL
LIN {X 0,Y 404.715,Z 1201.336,A -85,B 0,C 180,E1 17181.41,E2 17181.41} C_VEL
LIN {X 0,Y 404.474,Z 1205.429,A -85,B 0,C 180,E1 17187.858,E2 17187.858} C_VEL
LIN {X 0,Y 404.675,Z 1205.42,A -85,B 0,C 180,E1 17192.139,E2 17192.139} C_VEL
LIN {X 0,Y 404.713,Z 1201.235,A -85,B 0,C 180,E1 17198.588,E2 17198.588} C_VEL
LIN {X 0,Y 405.711,Z 1191.751,A -85,B 0,C 180,E1 17205.112,E2 17205.112} C_VEL
LIN {X 0,Y 408.609,Z 1176.998,A -85,B 0,C 180,E1 17211.704,E2 17211.704} C_VEL
LIN {X 0,Y 414.164,Z 1156.565,A -85,B 0,C 180,E1 17218.314,E2 17218.314} C_VEL
LIN {X 0,Y 416.16,Z 1150.403,A -85,B 0,C 180,E1 17219.949,E2 17219.949} C_VEL
LIN {X 0,Y 415.097,Z 1142.788,A -85,B 0,C 180,E1 17222.123,E2 17222.123} C_VEL
LIN {X 0,Y 414.431,Z 1134.544,A -85,B 0,C 180,E1 17224.262,E2 17224.262} C_VEL
LIN {X 0,Y 427.404,Z 1101.408,A -85,B 0,C 180,E1 17230.687,E2 17230.687} C_VEL
LIN {X 0,Y 441.132,Z 1067.268,A -85,B 0,C 180,E1 17235.679,E2 17235.679} C_VEL
LIN {X 0,Y 456.236,Z 1028.633,A -85,B 0,C 180,E1 17239.989,E2 17239.989} C_VEL
LIN {X 0,Y 471.139,Z 986.401,A -85,B 0,C 180,E1 17243.521,E2 17243.521} C_VEL
LIN {X 0,Y 485.242,Z 940.604,A -85,B 0,C 180,E1 17246.317,E2 17246.317} C_VEL
LIN {X 0,Y 494.802,Z 903.19,A -85,B 0,C 180,E1 17247.959,E2 17247.959} C_VEL
LIN {X 0,Y 487.676,Z 881.356,A -85,B 0,C 180,E1 17251.115,E2 17251.115} C_VEL
LIN {X 0,Y 476.559,Z 857.784,A -85,B 0,C 180,E1 17255.661,E2 17255.661} C_VEL
LIN {X 0,Y 466.71,Z 839.986,A -85,B 0,C 180,E1 17260.256,E2 17260.256} C_VEL
LIN {X 0,Y 459.601,Z 828.56,A -85,B 0,C 180,E1 17264.279,E2 17264.279} C_VEL
LIN {X 0,Y 456.342,Z 823.573,A -85,B 0,C 180,E1 17266.602,E2 17266.602} C_VEL
LIN {X 0,Y 453.414,Z 818.448,A -85,B 0,C 180,E1 17269.321,E2 17269.321} C_VEL
LIN {X 0,Y 450.28,Z 811.959,A -85,B 0,C 180,E1 17274.227,E2 17274.227} C_VEL
LIN {X 0,Y 450.453,Z 812.61,A -85,B 0,C 180,E1 17281.988,E2 17281.988} C_VEL
LIN {X 0,Y 453.606,Z 818.601,A -85,B 0,C 180,E1 17286.701,E2 17286.701} C_VEL
LIN {X 0,Y 458.838,Z 828.262,A -85,B 0,C 180,E1 17291.222,E2 17291.222} C_VEL
LIN {X 0,Y 465.174,Z 839.331,A -85,B 0,C 180,E1 17295.25,E2 17295.25} C_VEL
LIN {X 0,Y 474.22,Z 857.191,A -85,B 0,C 180,E1 17300.038,E2 17300.038} C_VEL
LIN {X 0,Y 483.776,Z 880.243,A -85,B 0,C 180,E1 17304.775,E2 17304.775} C_VEL
LIN {X 0,Y 489.34,Z 897.729,A -85,B 0,C 180,E1 17307.726,E2 17307.726} C_VEL
LIN {X 0,Y 476.924,Z 941.096,A -85,B 0,C 180,E1 17310.302,E2 17310.302} C_VEL
LIN {X 0,Y 461.919,Z 982.214,A -85,B 0,C 180,E1 17313.608,E2 17313.608} C_VEL
LIN {X 0,Y 447.415,Z 1017.374,A -85,B 0,C 180,E1 17317.449,E2 17317.449} C_VEL
LIN {X 0,Y 432.04,Z 1051.482,A -85,B 0,C 180,E1 17322.491,E2 17322.491} C_VEL
LIN {X 0,Y 419.179,Z 1079.147,A -85,B 0,C 180,E1 17328.083,E2 17328.083} C_VEL
LIN {X 0,Y 409.647,Z 1100.416,A -85,B 0,C 180,E1 17333.829,E2 17333.829} C_VEL
LIN {X 0,Y 402.384,Z 1118.746,A -85,B 0,C 180,E1 17340.778,E2 17340.778} C_VEL
LIN {X 0,Y 399.023,Z 1129.361,A -85,B 0,C 180,E1 17346.57,E2 17346.57} C_VEL
LIN {X 0,Y 397.34,Z 1136.144,A -85,B 0,C 180,E1 17352.288,E2 17352.288} C_VEL
LIN {X 0,Y 396.531,Z 1139.578,A -85,B 0,C 180,E1 17359.017,E2 17359.017} C_VEL
LIN {X 0,Y 396.941,Z 1138.351,A -85,B 0,C 180,E1 17365.634,E2 17365.634} C_VEL
LIN {X 0,Y 397.984,Z 1132.498,A -85,B 0,C 180,E1 17372.177,E2 17372.177} C_VEL
LIN {X 0,Y 400.478,Z 1121.875,A -85,B 0,C 180,E1 17378.682,E2 17378.682} C_VEL
LIN {X 0,Y 405.473,Z 1106.126,A -85,B 0,C 180,E1 17385.123,E2 17385.123} C_VEL
LIN {X 0,Y 414.136,Z 1083.392,A -85,B 0,C 180,E1 17391.683,E2 17391.683} C_VEL
LIN {X 0,Y 425.499,Z 1055.447,A -85,B 0,C 180,E1 17397.497,E2 17397.497} C_VEL
LIN {X 0,Y 438.02,Z 1024.36,A -85,B 0,C 180,E1 17402.33,E2 17402.33} C_VEL
LIN {X 0,Y 452.234,Z 986.255,A -85,B 0,C 180,E1 17406.741,E2 17406.741} C_VEL
LIN {X 0,Y 465.281,Z 946.349,A -85,B 0,C 180,E1 17410.118,E2 17410.118} C_VEL
LIN {X 0,Y 476.327,Z 906.295,A -85,B 0,C 180,E1 17412.649,E2 17412.649} C_VEL
LIN {X 0,Y 479.098,Z 893.394,A -85,B 0,C 180,E1 17413.339,E2 17413.339} C_VEL
LIN {X 0,Y 467.382,Z 861.417,A -85,B 0,C 180,E1 17417.857,E2 17417.857} C_VEL
LIN {X 0,Y 454.085,Z 833.492,A -85,B 0,C 180,E1 17422.507,E2 17422.507} C_VEL
LIN {X 0,Y 440.76,Z 811.009,A -85,B 0,C 180,E1 17427.237,E2 17427.237} C_VEL
LIN {X 0,Y 428.551,Z 792.913,A -85,B 0,C 180,E1 17432.145,E2 17432.145} C_VEL
LIN {X 0,Y 422.78,Z 785.507,A -85,B 0,C 180,E1 17434.845,E2 17434.845} C_VEL
LIN {X 0,Y 418.317,Z 779.29,A -85,B 0,C 180,E1 17437.283,E2 17437.283} C_VEL
LIN {X 0,Y 414.201,Z 773.298,A -85,B 0,C 180,E1 17439.993,E2 17439.993} C_VEL
LIN {X 0,Y 408.985,Z 767.037,A -85,B 0,C 180,E1 17444.574,E2 17444.574} C_VEL
LIN {X 0,Y 408.311,Z 765.069,A -85,B 0,C 180,E1 17445.527,E2 17445.527} C_VEL
LIN {X 0,Y 405.459,Z 763.096,A -85,B 0,C 180,E1 17454.648,E2 17454.648} C_VEL
LIN {X 0,Y 409.664,Z 765.918,A -85,B 0,C 180,E1 17461.712,E2 17461.712} C_VEL
LIN {X 0,Y 412.78,Z 771.424,A -85,B 0,C 180,E1 17464.686,E2 17464.686} C_VEL
LIN {X 0,Y 415.353,Z 773.869,A -85,B 0,C 180,E1 17466.506,E2 17466.506} C_VEL
LIN {X 0,Y 419.741,Z 779.648,A -85,B 0,C 180,E1 17469.206,E2 17469.206} C_VEL
LIN {X 0,Y 426.959,Z 790.067,A -85,B 0,C 180,E1 17472.839,E2 17472.839} C_VEL
LIN {X 0,Y 435.945,Z 802.321,A -85,B 0,C 180,E1 17476.482,E2 17476.482} C_VEL
LIN {X 0,Y 450.517,Z 824.41,A -85,B 0,C 180,E1 17481.453,E2 17481.453} C_VEL
LIN {X 0,Y 466.157,Z 852.755,A -85,B 0,C 180,E1 17486.271,E2 17486.271} C_VEL
LIN {X 0,Y 480.869,Z 885.135,A -85,B 0,C 180,E1 17490.704,E2 17490.704} C_VEL
LIN {X 0,Y 487.036,Z 900.674,A -85,B 0,C 180,E1 17492.643,E2 17492.643} C_VEL
LIN {X 0,Y 476.521,Z 947.261,A -85,B 0,C 180,E1 17494.765,E2 17494.765} C_VEL
LIN {X 0,Y 463.647,Z 993.522,A -85,B 0,C 180,E1 17497.702,E2 17497.702} C_VEL
LIN {X 0,Y 449.437,Z 1036.803,A -85,B 0,C 180,E1 17501.459,E2 17501.459} C_VEL
LIN {X 0,Y 436.201,Z 1074.085,A -85,B 0,C 180,E1 17505.733,E2 17505.733} C_VEL
LIN {X 0,Y 423.215,Z 1108.849,A -85,B 0,C 180,E1 17510.992,E2 17510.992} C_VEL
LIN {X 0,Y 412.694,Z 1137.749,A -85,B 0,C 180,E1 17516.684,E2 17516.684} C_VEL
LIN {X 0,Y 405.048,Z 1161.256,A -85,B 0,C 180,E1 17522.804,E2 17522.804} C_VEL
LIN {X 0,Y 400.036,Z 1180.673,A -85,B 0,C 180,E1 17529.547,E2 17529.547} C_VEL
LIN {X 0,Y 397.569,Z 1193.791,A -85,B 0,C 180,E1 17536.079,E2 17536.079} C_VEL
LIN {X 0,Y 396.736,Z 1201.32,A -85,B 0,C 180,E1 17541.985,E2 17541.985} C_VEL
LIN {X 0,Y 396.592,Z 1204.78,A -85,B 0,C 180,E1 17547.815,E2 17547.815} C_VEL
LIN {X 0,Y 396.786,Z 1204.768,A -85,B 0,C 180,E1 17552.181,E2 17552.181} C_VEL
LIN {X 0,Y 396.843,Z 1200.576,A -85,B 0,C 180,E1 17558.76,E2 17558.76} C_VEL
LIN {X 0,Y 397.907,Z 1191.091,A -85,B 0,C 180,E1 17565.416,E2 17565.416} C_VEL
LIN {X 0,Y 400.978,Z 1176.352,A -85,B 0,C 180,E1 17572.138,E2 17572.138} C_VEL
LIN {X 0,Y 406.848,Z 1155.953,A -85,B 0,C 180,E1 17578.87,E2 17578.87} C_VEL
LIN {X 0,Y 414.431,Z 1134.544,A -85,B 0,C 180,E1 17584.262,E2 17584.262} C_VEL
LIN {X 0,Y 414.127,Z 1126.079,A -85,B 0,C 180,E1 17586.378,E2 17586.378} C_VEL
LIN {X 0,Y 414.291,Z 1117.135,A -85,B 0,C 180,E1 17588.47,E2 17588.47} C_VEL
LIN {X 0,Y 427.562,Z 1085.59,A -85,B 0,C 180,E1 17593.876,E2 17593.876} C_VEL
LIN {X 0,Y 443.449,Z 1046.909,A -85,B 0,C 180,E1 17598.866,E2 17598.866} C_VEL
LIN {X 0,Y 459.193,Z 1006.567,A -85,B 0,C 180,E1 17602.745,E2 17602.745} C_VEL
LIN {X 0,Y 473.877,Z 963.81,A -85,B 0,C 180,E1 17605.781,E2 17605.781} C_VEL
LIN {X 0,Y 486.171,Z 921.287,A -85,B 0,C 180,E1 17608.011,E2 17608.011} C_VEL
LIN {X 0,Y 489.752,Z 905.874,A -85,B 0,C 180,E1 17608.683,E2 17608.683} C_VEL
LIN {X 0,Y 481.681,Z 882.294,A -85,B 0,C 180,E1 17612.384,E2 17612.384} C_VEL
LIN {X 0,Y 470.707,Z 858.977,A -85,B 0,C 180,E1 17617.284,E2 17617.284} C_VEL
LIN {X 0,Y 461.849,Z 843.202,A -85,B 0,C 180,E1 17621.827,E2 17621.827} C_VEL
LIN {X 0,Y 455.318,Z 832.125,A -85,B 0,C 180,E1 17626.207,E2 17626.207} C_VEL
LIN {X 0,Y 451.686,Z 826.042,A -85,B 0,C 180,E1 17629.524,E2 17629.524} C_VEL
LIN {X 0,Y 448.651,Z 819.669,A -85,B 0,C 180,E1 17634.691,E2 17634.691} C_VEL
LIN {X 0,Y 448.884,Z 820.402,A -85,B 0,C 180,E1 17641.874,E2 17641.874} C_VEL
LIN {X 0,Y 452.695,Z 828.079,A -85,B 0,C 180,E1 17647.438,E2 17647.438} C_VEL
LIN {X 0,Y 456.874,Z 836.138,A -85,B 0,C 180,E1 17651.21,E2 17651.21} C_VEL
LIN {X 0,Y 463.518,Z 848.476,A -85,B 0,C 180,E1 17655.608,E2 17655.608} C_VEL
LIN {X 0,Y 471.792,Z 865.864,A -85,B 0,C 180,E1 17660.226,E2 17660.226} C_VEL
LIN {X 0,Y 481.124,Z 890.524,A -85,B 0,C 180,E1 17665.197,E2 17665.197} C_VEL
LIN {X 0,Y 484.101,Z 903.335,A -85,B 0,C 180,E1 17667.234,E2 17667.234} C_VEL
LIN {X 0,Y 471.47,Z 944.401,A -85,B 0,C 180,E1 17669.695,E2 17669.695} C_VEL
LIN {X 0,Y 455.764,Z 986.055,A -85,B 0,C 180,E1 17673.125,E2 17673.125} C_VEL
LIN {X 0,Y 440.885,Z 1020.426,A -85,B 0,C 180,E1 17676.988,E2 17676.988} C_VEL
LIN {X 0,Y 425.83,Z 1052.586,A -85,B 0,C 180,E1 17681.824,E2 17681.824} C_VEL
LIN {X 0,Y 412.739,Z 1079.56,A -85,B 0,C 180,E1 17687.343,E2 17687.343} C_VEL
LIN {X 0,Y 402.291,Z 1101.882,A -85,B 0,C 180,E1 17693.49,E2 17693.49} C_VEL
LIN {X 0,Y 394.67,Z 1120.199,A -85,B 0,C 180,E1 17700.673,E2 17700.673} C_VEL
LIN {X 0,Y 390.919,Z 1131.493,A -85,B 0,C 180,E1 17707.261,E2 17707.261} C_VEL
LIN {X 0,Y 389.076,Z 1138.369,A -85,B 0,C 180,E1 17714.225,E2 17714.225} C_VEL
LIN {X 0,Y 388.689,Z 1140.386,A -85,B 0,C 180,E1 17721.055,E2 17721.055} C_VEL
LIN {X 0,Y 389.318,Z 1137.629,A -85,B 0,C 180,E1 17727.777,E2 17727.777} C_VEL
LIN {X 0,Y 390.353,Z 1131.884,A -85,B 0,C 180,E1 17733.33,E2 17733.33} C_VEL
LIN {X 0,Y 393.455,Z 1120.649,A -85,B 0,C 180,E1 17739.953,E2 17739.953} C_VEL
LIN {X 0,Y 399.744,Z 1102.353,A -85,B 0,C 180,E1 17747.037,E2 17747.037} C_VEL
LIN {X 0,Y 408.707,Z 1080.205,A -85,B 0,C 180,E1 17753.133,E2 17753.133} C_VEL
LIN {X 0,Y 420.401,Z 1052.71,A -85,B 0,C 180,E1 17758.736,E2 17758.736} C_VEL
LIN {X 0,Y 433.698,Z 1020.255,A -85,B 0,C 180,E1 17763.634,E2 17763.634} C_VEL
LIN {X 0,Y 447.531,Z 983.942,A -85,B 0,C 180,E1 17767.736,E2 17767.736} C_VEL
LIN {X 0,Y 461.441,Z 942.183,A -85,B 0,C 180,E1 17771.197,E2 17771.197} C_VEL
LIN {X 0,Y 472.533,Z 901.783,A -85,B 0,C 180,E1 17773.642,E2 17773.642} C_VEL
LIN {X 0,Y 473.527,Z 897.097,A -85,B 0,C 180,E1 17773.899,E2 17773.899} C_VEL
LIN {X 0,Y 462.504,Z 865.83,A -85,B 0,C 180,E1 17778.444,E2 17778.444} C_VEL
LIN {X 0,Y 449.747,Z 838.325,A -85,B 0,C 180,E1 17783.202,E2 17783.202} C_VEL
LIN {X 0,Y 437.564,Z 817.219,A -85,B 0,C 180,E1 17787.775,E2 17787.775} C_VEL
LIN {X 0,Y 426.327,Z 800.048,A -85,B 0,C 180,E1 17792.555,E2 17792.555} C_VEL
LIN {X 0,Y 420.856,Z 792.704,A -85,B 0,C 180,E1 17795.224,E2 17795.224} C_VEL
LIN {X 0,Y 416.721,Z 786.75,A -85,B 0,C 180,E1 17797.615,E2 17797.615} C_VEL
LIN {X 0,Y 411.645,Z 779.847,A -85,B 0,C 180,E1 17801.119,E2 17801.119} C_VEL
LIN {X 0,Y 407.602,Z 774.071,A -85,B 0,C 180,E1 17805.09,E2 17805.09} C_VEL
LIN {X 0,Y 406.511,Z 772.608,A -85,B 0,C 180,E1 17806.559,E2 17806.559} C_VEL
LIN {X 0,Y 404.489,Z 770.935,A -85,B 0,C 180,E1 17814.635,E2 17814.635} C_VEL
LIN {X 0,Y 408.453,Z 773.758,A -85,B 0,C 180,E1 17821.495,E2 17821.495} C_VEL
LIN {X 0,Y 412.022,Z 779.466,A -85,B 0,C 180,E1 17824.86,E2 17824.86} C_VEL
LIN {X 0,Y 414.046,Z 781.806,A -85,B 0,C 180,E1 17826.33,E2 17826.33} C_VEL
LIN {X 0,Y 419.746,Z 789.901,A -85,B 0,C 180,E1 17829.826,E2 17829.826} C_VEL
LIN {X 0,Y 425.229,Z 797.478,A -85,B 0,C 180,E1 17832.548,E2 17832.548} C_VEL
LIN {X 0,Y 436.783,Z 813.783,A -85,B 0,C 180,E1 17837.291,E2 17837.291} C_VEL
LIN {X 0,Y 451.983,Z 838.927,A -85,B 0,C 180,E1 17842.542,E2 17842.542} C_VEL
LIN {X 0,Y 466.745,Z 868.287,A -85,B 0,C 180,E1 17847.274,E2 17847.274} C_VEL
LIN {X 0,Y 481.499,Z 904.387,A -85,B 0,C 180,E1 17852.072,E2 17852.072} C_VEL
LIN {X 0,Y 469.898,Z 952.467,A -85,B 0,C 180,E1 17854.326,E2 17854.326} C_VEL
LIN {X 0,Y 457.088,Z 996.331,A -85,B 0,C 180,E1 17857.206,E2 17857.206} C_VEL
LIN {X 0,Y 441.95,Z 1041.062,A -85,B 0,C 180,E1 17861.215,E2 17861.215} C_VEL
LIN {X 0,Y 427.963,Z 1078.44,A -85,B 0,C 180,E1 17865.707,E2 17865.707} C_VEL
LIN {X 0,Y 414.528,Z 1113.61,A -85,B 0,C 180,E1 17871.284,E2 17871.284} C_VEL
LIN {X 0,Y 403.29,Z 1143.634,A -85,B 0,C 180,E1 17877.677,E2 17877.677} C_VEL
LIN {X 0,Y 395.785,Z 1166.776,A -85,B 0,C 180,E1 17884.256,E2 17884.256} C_VEL
LIN {X 0,Y 391.201,Z 1184.864,A -85,B 0,C 180,E1 17891.367,E2 17891.367} C_VEL
LIN {X 0,Y 389.281,Z 1195.889,A -85,B 0,C 180,E1 17897.671,E2 17897.671} C_VEL
LIN {X 0,Y 388.747,Z 1201.879,A -85,B 0,C 180,E1 17903.302,E2 17903.302} C_VEL
LIN {X 0,Y 388.896,Z 1204.491,A -85,B 0,C 180,E1 17909.999,E2 17909.999} C_VEL
LIN {X 0,Y 388.699,Z 1203.216,A -85,B 0,C 180,E1 17914.458,E2 17914.458} C_VEL
LIN {X 0,Y 389.038,Z 1198.616,A -85,B 0,C 180,E1 17920.065,E2 17920.065} C_VEL
LIN {X 0,Y 390.497,Z 1188.362,A -85,B 0,C 180,E1 17926.871,E2 17926.871} C_VEL
LIN {X 0,Y 394.158,Z 1172.654,A -85,B 0,C 180,E1 17933.798,E2 17933.798} C_VEL
LIN {X 0,Y 401.408,Z 1150.152,A -85,B 0,C 180,E1 17940.88,E2 17940.88} C_VEL
LIN {X 0,Y 411.738,Z 1123.262,A -85,B 0,C 180,E1 17947.269,E2 17947.269} C_VEL
LIN {X 0,Y 414.291,Z 1117.135,A -85,B 0,C 180,E1 17948.47,E2 17948.47} C_VEL
LIN {X 0,Y 414.9,Z 1107.926,A -85,B 0,C 180,E1 17950.529,E2 17950.529} C_VEL
LIN {X 0,Y 415.722,Z 1098.368,A -85,B 0,C 180,E1 17952.559,E2 17952.559} C_VEL
LIN {X 0,Y 431.823,Z 1061.34,A -85,B 0,C 180,E1 17957.926,E2 17957.926} C_VEL
LIN {X 0,Y 447.818,Z 1023.096,A -85,B 0,C 180,E1 17962.077,E2 17962.077} C_VEL
LIN {X 0,Y 463.849,Z 979.989,A -85,B 0,C 180,E1 17965.549,E2 17965.549} C_VEL
LIN {X 0,Y 477.873,Z 935.613,A -85,B 0,C 180,E1 17968.169,E2 17968.169} C_VEL
LIN {X 0,Y 484.706,Z 909.273,A -85,B 0,C 180,E1 17969.372,E2 17969.372} C_VEL
LIN {X 0,Y 476.911,Z 886.262,A -85,B 0,C 180,E1 17973.163,E2 17973.163} C_VEL
LIN {X 0,Y 466.491,Z 863.317,A -85,B 0,C 180,E1 17978.196,E2 17978.196} C_VEL
LIN {X 0,Y 457.161,Z 846.015,A -85,B 0,C 180,E1 17983.57,E2 17983.57} C_VEL
LIN {X 0,Y 452.355,Z 838.133,A -85,B 0,C 180,E1 17987.234,E2 17987.234} C_VEL
LIN {X 0,Y 449.96,Z 833.654,A -85,B 0,C 180,E1 17989.728,E2 17989.728} C_VEL
LIN {X 0,Y 446.966,Z 827.392,A -85,B 0,C 180,E1 17995.157,E2 17995.157} C_VEL
LIN {X 0,Y 447.32,Z 828.164,A -85,B 0,C 180,E1 18001.76,E2 18001.76} C_VEL
LIN {X 0,Y 450.653,Z 835.667,A -85,B 0,C 180,E1 18007.29,E2 18007.29} C_VEL
LIN {X 0,Y 455.387,Z 844.785,A -85,B 0,C 180,E1 18011.551,E2 18011.551} C_VEL
LIN {X 0,Y 462.673,Z 859.515,A -85,B 0,C 180,E1 18016.536,E2 18016.536} C_VEL
LIN {X 0,Y 471.611,Z 880.948,A -85,B 0,C 180,E1 18021.802,E2 18021.802} C_VEL
LIN {X 0,Y 478.923,Z 904.271,A -85,B 0,C 180,E1 18026.221,E2 18026.221} C_VEL
LIN {X 0,Y 478.686,Z 908.777,A -85,B 0,C 180,E1 18026.665,E2 18026.665} C_VEL
LIN {X 0,Y 464.688,Z 951.417,A -85,B 0,C 180,E1 18029.342,E2 18029.342} C_VEL
LIN {X 0,Y 449.721,Z 989.483,A -85,B 0,C 180,E1 18032.586,E2 18032.586} C_VEL
LIN {X 0,Y 433.198,Z 1026.111,A -85,B 0,C 180,E1 18036.87,E2 18036.87} C_VEL
LIN {X 0,Y 418.735,Z 1055.578,A -85,B 0,C 180,E1 18041.487,E2 18041.487} C_VEL
LIN {X 0,Y 404.14,Z 1084.587,A -85,B 0,C 180,E1 18047.699,E2 18047.699} C_VEL
LIN {X 0,Y 393.44,Z 1106.279,A -85,B 0,C 180,E1 18054.182,E2 18054.182} C_VEL
LIN {X 0,Y 386.796,Z 1122.092,A -85,B 0,C 180,E1 18060.769,E2 18060.769} C_VEL
LIN {X 0,Y 382.885,Z 1133.213,A -85,B 0,C 180,E1 18067.776,E2 18067.776} C_VEL
LIN {X 0,Y 381.259,Z 1138.934,A -85,B 0,C 180,E1 18073.893,E2 18073.893} C_VEL
LIN {X 0,Y 380.804,Z 1141.062,A -85,B 0,C 180,E1 18080.868,E2 18080.868} C_VEL
LIN {X 0,Y 381.457,Z 1138.376,A -85,B 0,C 180,E1 18087.731,E2 18087.731} C_VEL
LIN {X 0,Y 382.535,Z 1132.714,A -85,B 0,C 180,E1 18093.398,E2 18093.398} C_VEL
LIN {X 0,Y 385.732,Z 1121.587,A -85,B 0,C 180,E1 18100.155,E2 18100.155} C_VEL
LIN {X 0,Y 392.267,Z 1103.414,A -85,B 0,C 180,E1 18107.372,E2 18107.372} C_VEL
LIN {X 0,Y 401.539,Z 1081.429,A -85,B 0,C 180,E1 18113.57,E2 18113.57} C_VEL
LIN {X 0,Y 414.22,Z 1052.681,A -85,B 0,C 180,E1 18119.506,E2 18119.506} C_VEL
LIN {X 0,Y 428.664,Z 1018.523,A -85,B 0,C 180,E1 18124.643,E2 18124.643} C_VEL
LIN {X 0,Y 442.713,Z 982.25,A -85,B 0,C 180,E1 18128.688,E2 18128.688} C_VEL
LIN {X 0,Y 456.767,Z 941.119,A -85,B 0,C 180,E1 18132.063,E2 18132.063} C_VEL
LIN {X 0,Y 467.826,Z 900.367,A -85,B 0,C 180,E1 18134.541,E2 18134.541} C_VEL
LIN {X 0,Y 457.142,Z 869.134,A -85,B 0,C 180,E1 18139.235,E2 18139.235} C_VEL
LIN {X 0,Y 444.571,Z 841.443,A -85,B 0,C 180,E1 18144.221,E2 18144.221} C_VEL
LIN {X 0,Y 432.197,Z 819.729,A -85,B 0,C 180,E1 18149.239,E2 18149.239} C_VEL
LIN {X 0,Y 420.673,Z 801.642,A -85,B 0,C 180,E1 18154.71,E2 18154.71} C_VEL
LIN {X 0,Y 414.807,Z 794.005,A -85,B 0,C 180,E1 18158.071,E2 18158.071} C_VEL
LIN {X 0,Y 410.543,Z 787.626,A -85,B 0,C 180,E1 18161.205,E2 18161.205} C_VEL
LIN {X 0,Y 406.479,Z 781.869,A -85,B 0,C 180,E1 18165.254,E2 18165.254} C_VEL
LIN {X 0,Y 405.01,Z 780.179,A -85,B 0,C 180,E1 18167.342,E2 18167.342} C_VEL
LIN {X 0,Y 403.801,Z 778.892,A -85,B 0,C 180,E1 18175.702,E2 18175.702} C_VEL
LIN {X 0,Y 407.273,Z 781.607,A -85,B 0,C 180,E1 18181.302,E2 18181.302} C_VEL
LIN {X 0,Y 411.271,Z 787.473,A -85,B 0,C 180,E1 18185.034,E2 18185.034} C_VEL
LIN {X 0,Y 418.233,Z 797.455,A -85,B 0,C 180,E1 18189.577,E2 18189.577} C_VEL
LIN {X 0,Y 426.751,Z 809.474,A -85,B 0,C 180,E1 18193.794,E2 18193.794} C_VEL
LIN {X 0,Y 439.072,Z 828.719,A -85,B 0,C 180,E1 18198.753,E2 18198.753} C_VEL
LIN {X 0,Y 452.874,Z 853.461,A -85,B 0,C 180,E1 18203.599,E2 18203.599} C_VEL
LIN {X 0,Y 467.291,Z 885.266,A -85,B 0,C 180,E1 18208.463,E2 18208.463} C_VEL
LIN {X 0,Y 475.727,Z 907.959,A -85,B 0,C 180,E1 18211.465,E2 18211.465} C_VEL
LIN {X 0,Y 463.683,Z 956.337,A -85,B 0,C 180,E1 18213.805,E2 18213.805} C_VEL
LIN {X 0,Y 450.218,Z 1000.149,A -85,B 0,C 180,E1 18216.784,E2 18216.784} C_VEL
LIN {X 0,Y 435.766,Z 1041.42,A -85,B 0,C 180,E1 18220.556,E2 18220.556} C_VEL
LIN {X 0,Y 421.885,Z 1077.395,A -85,B 0,C 180,E1 18224.926,E2 18224.926} C_VEL
LIN {X 0,Y 408.34,Z 1111.406,A -85,B 0,C 180,E1 18230.329,E2 18230.329} C_VEL
LIN {X 0,Y 397.291,Z 1139.574,A -85,B 0,C 180,E1 18236.257,E2 18236.257} C_VEL
LIN {X 0,Y 389.047,Z 1163.471,A -85,B 0,C 180,E1 18242.906,E2 18242.906} C_VEL
LIN {X 0,Y 384.081,Z 1181.507,A -85,B 0,C 180,E1 18249.757,E2 18249.757} C_VEL
LIN {X 0,Y 381.723,Z 1193.495,A -85,B 0,C 180,E1 18256.258,E2 18256.258} C_VEL
LIN {X 0,Y 380.876,Z 1200.792,A -85,B 0,C 180,E1 18262.653,E2 18262.653} C_VEL
LIN {X 0,Y 380.828,Z 1203.476,A -85,B 0,C 180,E1 18267.725,E2 18267.725} C_VEL
LIN {X 0,Y 381.008,Z 1203.468,A -85,B 0,C 180,E1 18272.272,E2 18272.272} C_VEL
LIN {X 0,Y 381.076,Z 1199.279,A -85,B 0,C 180,E1 18279.125,E2 18279.125} C_VEL
LIN {X 0,Y 382.337,Z 1189.812,A -85,B 0,C 180,E1 18286.06,E2 18286.06} C_VEL
LIN {X 0,Y 385.71,Z 1175.094,A -85,B 0,C 180,E1 18293.064,E2 18293.064} C_VEL
LIN {X 0,Y 392.379,Z 1154.782,A -85,B 0,C 180,E1 18300.042,E2 18300.042} C_VEL
LIN {X 0,Y 402.942,Z 1127.83,A -85,B 0,C 180,E1 18306.871,E2 18306.871} C_VEL
LIN {X 0,Y 415.722,Z 1098.368,A -85,B 0,C 180,E1 18312.559,E2 18312.559} C_VEL
LIN {X 0,Y 416.926,Z 1088.428,A -85,B 0,C 180,E1 18314.549,E2 18314.549} C_VEL
LIN {X 0,Y 418.072,Z 1079.392,A -85,B 0,C 180,E1 18316.246,E2 18316.246} C_VEL
LIN {X 0,Y 418.686,Z 1077.954,A -85,B 0,C 180,E1 18316.457,E2 18316.457} C_VEL
LIN {X 0,Y 435.193,Z 1040.94,A -85,B 0,C 180,E1 18321.095,E2 18321.095} C_VEL
LIN {X 0,Y 452.387,Z 998.346,A -85,B 0,C 180,E1 18325.03,E2 18325.03} C_VEL
LIN {X 0,Y 467.978,Z 954.54,A -85,B 0,C 180,E1 18327.969,E2 18327.969} C_VEL
LIN {X 0,Y 479.825,Z 913.224,A -85,B 0,C 180,E1 18330.008,E2 18330.008} C_VEL
LIN {X 0,Y 473.256,Z 892.854,A -85,B 0,C 180,E1 18333.452,E2 18333.452} C_VEL
LIN {X 0,Y 463.365,Z 870.009,A -85,B 0,C 180,E1 18338.544,E2 18338.544} C_VEL
LIN {X 0,Y 454.774,Z 853.277,A -85,B 0,C 180,E1 18343.846,E2 18343.846} C_VEL
LIN {X 0,Y 448.551,Z 841.675,A -85,B 0,C 180,E1 18349.327,E2 18349.327} C_VEL
LIN {X 0,Y 445.359,Z 835.125,A -85,B 0,C 180,E1 18355.139,E2 18355.139} C_VEL
LIN {X 0,Y 445.493,Z 835.853,A -85,B 0,C 180,E1 18361.645,E2 18361.645} C_VEL
LIN {X 0,Y 448.617,Z 843.246,A -85,B 0,C 180,E1 18367.141,E2 18367.141} C_VEL
LIN {X 0,Y 452.897,Z 852.225,A -85,B 0,C 180,E1 18371.401,E2 18371.401} C_VEL
LIN {X 0,Y 459.5,Z 866.354,A -85,B 0,C 180,E1 18376.24,E2 18376.24} C_VEL
LIN {X 0,Y 467.408,Z 886.464,A -85,B 0,C 180,E1 18381.285,E2 18381.285} C_VEL
LIN {X 0,Y 474.414,Z 910.012,A -85,B 0,C 180,E1 18385.859,E2 18385.859} C_VEL
LIN {X 0,Y 459.739,Z 953.551,A -85,B 0,C 180,E1 18388.624,E2 18388.624} C_VEL
LIN {X 0,Y 444.072,Z 991.913,A -85,B 0,C 180,E1 18391.943,E2 18391.943} C_VEL
LIN {X 0,Y 427.113,Z 1028.315,A -85,B 0,C 180,E1 18396.27,E2 18396.27} C_VEL
LIN {X 0,Y 411.301,Z 1059.192,A -85,B 0,C 180,E1 18401.274,E2 18401.274} C_VEL
LIN {X 0,Y 397.232,Z 1086.022,A -85,B 0,C 180,E1 18407.182,E2 18407.182} C_VEL
LIN {X 0,Y 385.787,Z 1108.205,A -85,B 0,C 180,E1 18414.018,E2 18414.018} C_VEL
LIN {X 0,Y 378.98,Z 1123.637,A -85,B 0,C 180,E1 18420.763,E2 18420.763} C_VEL
LIN {X 0,Y 374.959,Z 1134.536,A -85,B 0,C 180,E1 18427.981,E2 18427.981} C_VEL
LIN {X 0,Y 373.443,Z 1139.501,A -85,B 0,C 180,E1 18433.547,E2 18433.547} C_VEL
LIN {X 0,Y 372.932,Z 1141.736,A -85,B 0,C 180,E1 18440.673,E2 18440.673} C_VEL
LIN {X 0,Y 373.57,Z 1139.124,A -85,B 0,C 180,E1 18447.683,E2 18447.683} C_VEL
LIN {X 0,Y 374.713,Z 1133.538,A -85,B 0,C 180,E1 18453.469,E2 18453.469} C_VEL
LIN {X 0,Y 378.022,Z 1122.502,A -85,B 0,C 180,E1 18460.364,E2 18460.364} C_VEL
LIN {X 0,Y 384.782,Z 1104.469,A -85,B 0,C 180,E1 18467.721,E2 18467.721} C_VEL
LIN {X 0,Y 394.382,Z 1082.647,A -85,B 0,C 180,E1 18474.025,E2 18474.025} C_VEL
LIN {X 0,Y 407.468,Z 1054.019,A -85,B 0,C 180,E1 18480.045,E2 18480.045} C_VEL
LIN {X 0,Y 421.519,Z 1021.887,A -85,B 0,C 180,E1 18485.002,E2 18485.002} C_VEL
LIN {X 0,Y 436.328,Z 985.298,A -85,B 0,C 180,E1 18489.203,E2 18489.203} C_VEL
LIN {X 0,Y 451.605,Z 941.791,A -85,B 0,C 180,E1 18492.82,E2 18492.82} C_VEL
LIN {X 0,Y 462.229,Z 903.718,A -85,B 0,C 180,E1 18495.183,E2 18495.183} C_VEL
LIN {X 0,Y 452.216,Z 873.286,A -85,B 0,C 180,E1 18499.902,E2 18499.902} C_VEL
LIN {X 0,Y 440.142,Z 846.149,A -85,B 0,C 180,E1 18504.958,E2 18504.958} C_VEL
LIN {X 0,Y 428.701,Z 825.441,A -85,B 0,C 180,E1 18509.946,E2 18509.946} C_VEL
LIN {X 0,Y 418.575,Z 808.944,A -85,B 0,C 180,E1 18515.08,E2 18515.08} C_VEL
LIN {X 0,Y 413.091,Z 801.436,A -85,B 0,C 180,E1 18518.396,E2 18518.396} C_VEL
LIN {X 0,Y 408.977,Z 795.187,A -85,B 0,C 180,E1 18521.549,E2 18521.549} C_VEL
LIN {X 0,Y 405.189,Z 789.091,A -85,B 0,C 180,E1 18525.688,E2 18525.688} C_VEL
LIN {X 0,Y 402.414,Z 786.481,A -85,B 0,C 180,E1 18533.525,E2 18533.525} C_VEL
LIN {X 0,Y 406.071,Z 789.287,A -85,B 0,C 180,E1 18541.06,E2 18541.06} C_VEL
LIN {X 0,Y 410.068,Z 795.227,A -85,B 0,C 180,E1 18544.883,E2 18544.883} C_VEL
LIN {X 0,Y 416.735,Z 805.325,A -85,B 0,C 180,E1 18549.426,E2 18549.426} C_VEL
LIN {X 0,Y 424.843,Z 816.951,A -85,B 0,C 180,E1 18553.525,E2 18553.525} C_VEL
LIN {X 0,Y 436.834,Z 836.482,A -85,B 0,C 180,E1 18558.591,E2 18558.591} C_VEL
LIN {X 0,Y 449.981,Z 861.144,A -85,B 0,C 180,E1 18563.432,E2 18563.432} C_VEL
LIN {X 0,Y 462.692,Z 890.718,A -85,B 0,C 180,E1 18568.045,E2 18568.045} C_VEL
LIN {X 0,Y 469.892,Z 912.168,A -85,B 0,C 180,E1 18570.877,E2 18570.877} C_VEL
LIN {X 0,Y 457.775,Z 958.995,A -85,B 0,C 180,E1 18573.206,E2 18573.206} C_VEL
LIN {X 0,Y 442.54,Z 1006.409,A -85,B 0,C 180,E1 18576.549,E2 18576.549} C_VEL
LIN {X 0,Y 427.991,Z 1045.851,A -85,B 0,C 180,E1 18580.333,E2 18580.333} C_VEL
LIN {X 0,Y 412.648,Z 1084.312,A -85,B 0,C 180,E1 18585.255,E2 18585.255} C_VEL
LIN {X 0,Y 399.287,Z 1116.507,A -85,B 0,C 180,E1 18590.748,E2 18590.748} C_VEL
LIN {X 0,Y 387.827,Z 1145.425,A -85,B 0,C 180,E1 18597.272,E2 18597.272} C_VEL
LIN {X 0,Y 380.075,Z 1167.607,A -85,B 0,C 180,E1 18604.064,E2 18604.064} C_VEL
LIN {X 0,Y 375.45,Z 1184.682,A -85,B 0,C 180,E1 18611.216,E2 18611.216} C_VEL
LIN {X 0,Y 373.614,Z 1194.469,A -85,B 0,C 180,E1 18617.146,E2 18617.146} C_VEL
LIN {X 0,Y 373.002,Z 1200.531,A -85,B 0,C 180,E1 18623.018,E2 18623.018} C_VEL
LIN {X 0,Y 373.142,Z 1203.187,A -85,B 0,C 180,E1 18629.999,E2 18629.999} C_VEL
LIN {X 0,Y 372.921,Z 1201.927,A -85,B 0,C 180,E1 18634.647,E2 18634.647} C_VEL
LIN {X 0,Y 373.281,Z 1197.336,A -85,B 0,C 180,E1 18640.495,E2 18640.495} C_VEL
LIN {X 0,Y 374.943,Z 1187.098,A -85,B 0,C 180,E1 18647.593,E2 18647.593} C_VEL
LIN {X 0,Y 379.061,Z 1171.61,A -85,B 0,C 180,E1 18654.744,E2 18654.744} C_VEL
LIN {X 0,Y 387.188,Z 1149.092,A -85,B 0,C 180,E1 18662.123,E2 18662.123} C_VEL
LIN {X 0,Y 398.942,Z 1121.389,A -85,B 0,C 180,E1 18668.898,E2 18668.898} C_VEL
LIN {X 0,Y 414.138,Z 1087.953,A -85,B 0,C 180,E1 18674.96,E2 18674.96} C_VEL
LIN {X 0,Y 418.686,Z 1077.954,A -85,B 0,C 180,E1 18676.457,E2 18676.457} C_VEL
LIN {X 0,Y 420.694,Z 1067.305,A -85,B 0,C 180,E1 18678.329,E2 18678.329} C_VEL
LIN {X 0,Y 422.283,Z 1057.741,A -85,B 0,C 180,E1 18679.961,E2 18679.961} C_VEL
LIN {X 0,Y 422.946,Z 1056.237,A -85,B 0,C 180,E1 18680.159,E2 18680.159} C_VEL
LIN {X 0,Y 440.286,Z 1016.696,A -85,B 0,C 180,E1 18684.311,E2 18684.311} C_VEL
LIN {X 0,Y 456.058,Z 976.571,A -85,B 0,C 180,E1 18687.442,E2 18687.442} C_VEL
LIN {X 0,Y 470.653,Z 932.18,A -85,B 0,C 180,E1 18689.982,E2 18689.982} C_VEL
LIN {X 0,Y 474.879,Z 916.89,A -85,B 0,C 180,E1 18690.714,E2 18690.714} C_VEL
LIN {X 0,Y 467.996,Z 895.346,A -85,B 0,C 180,E1 18694.565,E2 18694.565} C_VEL
LIN {X 0,Y 459.102,Z 874.522,A -85,B 0,C 180,E1 18699.535,E2 18699.535} C_VEL
LIN {X 0,Y 451.969,Z 860.068,A -85,B 0,C 180,E1 18704.305,E2 18704.305} C_VEL
LIN {X 0,Y 446.603,Z 849.307,A -85,B 0,C 180,E1 18709.402,E2 18709.402} C_VEL
LIN {X 0,Y 443.525,Z 842.788,A -85,B 0,C 180,E1 18715.119,E2 18715.119} C_VEL
LIN {X 0,Y 443.602,Z 843.482,A -85,B 0,C 180,E1 18721.53,E2 18721.53} C_VEL
LIN {X 0,Y 446.463,Z 851.051,A -85,B 0,C 180,E1 18727.114,E2 18727.114} C_VEL
LIN {X 0,Y 451.181,Z 860.921,A -85,B 0,C 180,E1 18731.844,E2 18731.844} C_VEL
LIN {X 0,Y 458.24,Z 877.85,A -85,B 0,C 180,E1 18737.271,E2 18737.271} C_VEL
LIN {X 0,Y 465.625,Z 899.632,A -85,B 0,C 180,E1 18742.422,E2 18742.422} C_VEL
LIN {X 0,Y 469.348,Z 913.85,A -85,B 0,C 180,E1 18745.177,E2 18745.177} C_VEL
LIN {X 0,Y 453.932,Z 958.261,A -85,B 0,C 180,E1 18748.086,E2 18748.086} C_VEL
LIN {X 0,Y 437.098,Z 997.399,A -85,B 0,C 180,E1 18751.609,E2 18751.609} C_VEL
LIN {X 0,Y 420.939,Z 1030.794,A -85,B 0,C 180,E1 18755.689,E2 18755.689} C_VEL
LIN {X 0,Y 403.984,Z 1062.516,A -85,B 0,C 180,E1 18760.988,E2 18760.988} C_VEL
LIN {X 0,Y 389.733,Z 1088.521,A -85,B 0,C 180,E1 18766.959,E2 18766.959} C_VEL
LIN {X 0,Y 377.708,Z 1111.041,A -85,B 0,C 180,E1 18774.183,E2 18774.183} C_VEL
LIN {X 0,Y 370.628,Z 1126.372,A -85,B 0,C 180,E1 18781.446,E2 18781.446} C_VEL
LIN {X 0,Y 367.034,Z 1135.926,A -85,B 0,C 180,E1 18788.252,E2 18788.252} C_VEL
LIN {X 0,Y 365.636,Z 1140.07,A -85,B 0,C 180,E1 18793.185,E2 18793.185} C_VEL
LIN {X 0,Y 365.042,Z 1142.396,A -85,B 0,C 180,E1 18800.47,E2 18800.47} C_VEL
LIN {X 0,Y 365.389,Z 1141.186,A -85,B 0,C 180,E1 18805.257,E2 18805.257} C_VEL
LIN {X 0,Y 366.641,Z 1135.813,A -85,B 0,C 180,E1 18812.363,E2 18812.363} C_VEL
LIN {X 0,Y 369.49,Z 1125.543,A -85,B 0,C 180,E1 18819.417,E2 18819.417} C_VEL
LIN {X 0,Y 375.321,Z 1110.321,A -85,B 0,C 180,E1 18826.371,E2 18826.371} C_VEL
LIN {X 0,Y 384.766,Z 1089.045,A -85,B 0,C 180,E1 18833.126,E2 18833.126} C_VEL
LIN {X 0,Y 397.304,Z 1062.705,A -85,B 0,C 180,E1 18839.2,E2 18839.2} C_VEL
LIN {X 0,Y 412.171,Z 1030.511,A -85,B 0,C 180,E1 18844.631,E2 18844.631} C_VEL
LIN {X 0,Y 427.2,Z 995.171,A -85,B 0,C 180,E1 18848.999,E2 18848.999} C_VEL
LIN {X 0,Y 441.721,Z 956.951,A -85,B 0,C 180,E1 18852.506,E2 18852.506} C_VEL
LIN {X 0,Y 455.107,Z 913.963,A -85,B 0,C 180,E1 18855.386,E2 18855.386} C_VEL
LIN {X 0,Y 456.724,Z 907.247,A -85,B 0,C 180,E1 18855.815,E2 18855.815} C_VEL
LIN {X 0,Y 447.559,Z 878.384,A -85,B 0,C 180,E1 18860.416,E2 18860.416} C_VEL
LIN {X 0,Y 435.807,Z 850.792,A -85,B 0,C 180,E1 18865.709,E2 18865.709} C_VEL
LIN {X 0,Y 425.01,Z 830.806,A -85,B 0,C 180,E1 18870.726,E2 18870.726} C_VEL
LIN {X 0,Y 416.054,Z 815.861,A -85,B 0,C 180,E1 18875.59,E2 18875.59} C_VEL
LIN {X 0,Y 411.041,Z 808.507,A -85,B 0,C 180,E1 18878.928,E2 18878.928} C_VEL
LIN {X 0,Y 407.383,Z 802.738,A -85,B 0,C 180,E1 18881.894,E2 18881.894} C_VEL
LIN {X 0,Y 403.564,Z 796.13,A -85,B 0,C 180,E1 18886.459,E2 18886.459} C_VEL
LIN {X 0,Y 401.847,Z 794.56,A -85,B 0,C 180,E1 18895.681,E2 18895.681} C_VEL
LIN {X 0,Y 404.878,Z 797.048,A -85,B 0,C 180,E1 18900.863,E2 18900.863} C_VEL
LIN {X 0,Y 408.954,Z 803.07,A -85,B 0,C 180,E1 18904.896,E2 18904.896} C_VEL
LIN {X 0,Y 418.374,Z 817.298,A -85,B 0,C 180,E1 18910.983,E2 18910.983} C_VEL
LIN {X 0,Y 429.819,Z 835.985,A -85,B 0,C 180,E1 18916.494,E2 18916.494} C_VEL
LIN {X 0,Y 443.13,Z 860.643,A -85,B 0,C 180,E1 18921.829,E2 18921.829} C_VEL
LIN {X 0,Y 455.915,Z 890.275,A -85,B 0,C 180,E1 18926.761,E2 18926.761} C_VEL
LIN {X 0,Y 464.466,Z 914.218,A -85,B 0,C 180,E1 18930.16,E2 18930.16} C_VEL
LIN {X 0,Y 452.535,Z 959.342,A -85,B 0,C 180,E1 18932.458,E2 18932.458} C_VEL
LIN {X 0,Y 436.959,Z 1006.59,A -85,B 0,C 180,E1 18935.81,E2 18935.81} C_VEL
LIN {X 0,Y 421.488,Z 1047.139,A -85,B 0,C 180,E1 18939.757,E2 18939.757} C_VEL
LIN {X 0,Y 406.06,Z 1084.552,A -85,B 0,C 180,E1 18944.623,E2 18944.623} C_VEL
LIN {X 0,Y 391.6,Z 1118.145,A -85,B 0,C 180,E1 18950.505,E2 18950.505} C_VEL
LIN {X 0,Y 380.233,Z 1145.798,A -85,B 0,C 180,E1 18956.946,E2 18956.946} C_VEL
LIN {X 0,Y 372.06,Z 1168.416,A -85,B 0,C 180,E1 18964.111,E2 18964.111} C_VEL
LIN {X 0,Y 367.641,Z 1184.219,A -85,B 0,C 180,E1 18970.959,E2 18970.959} C_VEL
LIN {X 0,Y 365.763,Z 1193.843,A -85,B 0,C 180,E1 18976.932,E2 18976.932} C_VEL
LIN {X 0,Y 365.064,Z 1200.253,A -85,B 0,C 180,E1 18983.391,E2 18983.391} C_VEL
LIN {X 0,Y 365.266,Z 1202.532,A -85,B 0,C 180,E1 18989.999,E2 18989.999} C_VEL
LIN {X 0,Y 365.058,Z 1200.328,A -85,B 0,C 180,E1 18996.601,E2 18996.601} C_VEL
LIN {X 0,Y 365.734,Z 1194.047,A -85,B 0,C 180,E1 19003.052,E2 19003.052} C_VEL
LIN {X 0,Y 368.327,Z 1181.894,A -85,B 0,C 180,E1 19010.408,E2 19010.408} C_VEL
LIN {X 0,Y 373.979,Z 1163.965,A -85,B 0,C 180,E1 19017.903,E2 19017.903} C_VEL
LIN {X 0,Y 383.194,Z 1141.061,A -85,B 0,C 180,E1 19024.874,E2 19024.874} C_VEL
LIN {X 0,Y 397.327,Z 1110.442,A -85,B 0,C 180,E1 19031.81,E2 19031.81} C_VEL
LIN {X 0,Y 413.89,Z 1075.613,A -85,B 0,C 180,E1 19037.579,E2 19037.579} C_VEL
LIN {X 0,Y 422.946,Z 1056.237,A -85,B 0,C 180,E1 19040.159,E2 19040.159} C_VEL
LIN {X 0,Y 425.633,Z 1044.807,A -85,B 0,C 180,E1 19041.92,E2 19041.92} C_VEL
LIN {X 0,Y 428.353,Z 1032.866,A -85,B 0,C 180,E1 19043.602,E2 19043.602} C_VEL
LIN {X 0,Y 446.052,Z 991.107,A -85,B 0,C 180,E1 19047.293,E2 19047.293} C_VEL
LIN {X 0,Y 461.97,Z 946.986,A -85,B 0,C 180,E1 19050.09,E2 19050.09} C_VEL
LIN {X 0,Y 469.942,Z 920.507,A -85,B 0,C 180,E1 19051.426,E2 19051.426} C_VEL
LIN {X 0,Y 463.232,Z 899.018,A -85,B 0,C 180,E1 19055.479,E2 19055.479} C_VEL
LIN {X 0,Y 454.861,Z 878.622,A -85,B 0,C 180,E1 19060.602,E2 19060.602} C_VEL
LIN {X 0,Y 447.327,Z 862.719,A -85,B 0,C 180,E1 19066.389,E2 19066.389} C_VEL
LIN {X 0,Y 443.55,Z 855.953,A -85,B 0,C 180,E1 19070.57,E2 19070.57} C_VEL
LIN {X 0,Y 441.689,Z 850.462,A -85,B 0,C 180,E1 19075.099,E2 19075.099} C_VEL
LIN {X 0,Y 441.607,Z 851.017,A -85,B 0,C 180,E1 19081.353,E2 19081.353} C_VEL
LIN {X 0,Y 444.087,Z 858.462,A -85,B 0,C 180,E1 19086.941,E2 19086.941} C_VEL
LIN {X 0,Y 448.392,Z 868.291,A -85,B 0,C 180,E1 19091.672,E2 19091.672} C_VEL
LIN {X 0,Y 454.802,Z 884.699,A -85,B 0,C 180,E1 19097.03,E2 19097.03} C_VEL
LIN {X 0,Y 461.372,Z 905.458,A -85,B 0,C 180,E1 19102.029,E2 19102.029} C_VEL
LIN {X 0,Y 464.123,Z 919.14,A -85,B 0,C 180,E1 19104.622,E2 19104.622} C_VEL
LIN {X 0,Y 449.052,Z 960.547,A -85,B 0,C 180,E1 19107.356,E2 19107.356} C_VEL
LIN {X 0,Y 431.655,Z 999.606,A -85,B 0,C 180,E1 19110.912,E2 19110.912} C_VEL
LIN {X 0,Y 415.085,Z 1032.602,A -85,B 0,C 180,E1 19115.007,E2 19115.007} C_VEL
LIN {X 0,Y 397.287,Z 1064.729,A -85,B 0,C 180,E1 19120.474,E2 19120.474} C_VEL
LIN {X 0,Y 382.841,Z 1089.964,A -85,B 0,C 180,E1 19126.427,E2 19126.427} C_VEL
LIN {X 0,Y 371.295,Z 1110.539,A -85,B 0,C 180,E1 19133.109,E2 19133.109} C_VEL
LIN {X 0,Y 363.779,Z 1125.603,A -85,B 0,C 180,E1 19140.102,E2 19140.102} C_VEL
LIN {X 0,Y 359.348,Z 1136.429,A -85,B 0,C 180,E1 19147.763,E2 19147.763} C_VEL
LIN {X 0,Y 357.421,Z 1141.958,A -85,B 0,C 180,E1 19155.306,E2 19155.306} C_VEL
LIN {X 0,Y 357.254,Z 1142.703,A -85,B 0,C 180,E1 19162.711,E2 19162.711} C_VEL
LIN {X 0,Y 358.281,Z 1138.861,A -85,B 0,C 180,E1 19170.001,E2 19170.001} C_VEL
LIN {X 0,Y 360.493,Z 1130.349,A -85,B 0,C 180,E1 19177.226,E2 19177.226} C_VEL
LIN {X 0,Y 365.311,Z 1117.023,A -85,B 0,C 180,E1 19184.372,E2 19184.372} C_VEL
LIN {X 0,Y 373.799,Z 1097.941,A -85,B 0,C 180,E1 19191.337,E2 19191.337} C_VEL
LIN {X 0,Y 385.153,Z 1074.854,A -85,B 0,C 180,E1 19197.453,E2 19197.453} C_VEL
LIN {X 0,Y 400.436,Z 1043.406,A -85,B 0,C 180,E1 19203.499,E2 19203.499} C_VEL
LIN {X 0,Y 415.719,Z 1009.927,A -85,B 0,C 180,E1 19208.168,E2 19208.168} C_VEL
LIN {X 0,Y 431.06,Z 972.38,A -85,B 0,C 180,E1 19212.073,E2 19212.073} C_VEL
LIN {X 0,Y 446.518,Z 927.432,A -85,B 0,C 180,E1 19215.431,E2 19215.431} C_VEL
LIN {X 0,Y 451.225,Z 911.014,A -85,B 0,C 180,E1 19216.417,E2 19216.417} C_VEL
LIN {X 0,Y 442.429,Z 882.201,A -85,B 0,C 180,E1 19221.162,E2 19221.162} C_VEL
LIN {X 0,Y 431.604,Z 855.771,A -85,B 0,C 180,E1 19226.427,E2 19226.427} C_VEL
LIN {X 0,Y 420.913,Z 835.191,A -85,B 0,C 180,E1 19231.789,E2 19231.789} C_VEL
LIN {X 0,Y 412.742,Z 821.585,A -85,B 0,C 180,E1 19236.623,E2 19236.623} C_VEL
LIN {X 0,Y 409.055,Z 815.891,A -85,B 0,C 180,E1 19239.237,E2 19239.237} C_VEL
LIN {X 0,Y 405.744,Z 810.248,A -85,B 0,C 180,E1 19242.239,E2 19242.239} C_VEL
LIN {X 0,Y 402.07,Z 803.772,A -85,B 0,C 180,E1 19246.961,E2 19246.961} C_VEL
LIN {X 0,Y 400.698,Z 802.376,A -85,B 0,C 180,E1 19255.668,E2 19255.668} C_VEL
LIN {X 0,Y 403.545,Z 804.789,A -85,B 0,C 180,E1 19260.665,E2 19260.665} C_VEL
LIN {X 0,Y 408.569,Z 812.917,A -85,B 0,C 180,E1 19265.61,E2 19265.61} C_VEL
LIN {X 0,Y 416.176,Z 824.498,A -85,B 0,C 180,E1 19270.65,E2 19270.65} C_VEL
LIN {X 0,Y 426.998,Z 842.805,A -85,B 0,C 180,E1 19276.114,E2 19276.114} C_VEL
LIN {X 0,Y 439.547,Z 867.248,A -85,B 0,C 180,E1 19281.486,E2 19281.486} C_VEL
LIN {X 0,Y 451.412,Z 895.747,A -85,B 0,C 180,E1 19286.319,E2 19286.319} C_VEL
LIN {X 0,Y 458.94,Z 917.795,A -85,B 0,C 180,E1 19289.524,E2 19289.524} C_VEL
LIN {X 0,Y 446.006,Z 963.976,A -85,B 0,C 180,E1 19291.958,E2 19291.958} C_VEL
LIN {X 0,Y 430.645,Z 1008.979,A -85,B 0,C 180,E1 19295.234,E2 19295.234} C_VEL
LIN {X 0,Y 414.033,Z 1050.742,A -85,B 0,C 180,E1 19299.428,E2 19299.428} C_VEL
LIN {X 0,Y 398.879,Z 1086.224,A -85,B 0,C 180,E1 19304.204,E2 19304.204} C_VEL
LIN {X 0,Y 383.363,Z 1121.192,A -85,B 0,C 180,E1 19310.547,E2 19310.547} C_VEL
